# B&R Automation Studio project perfxxl
Automation Studio 4.1.4.402

## Configuration Config1

CPU , AutomationRuntime A3.10, Build 2.95.3, Vc V4.14.1

### Task classes (Cpu.sw)
```
Cyclic#1 (cycle 1000 us, tolerance 40000 us):
  flow <- Processor.flow.prg
Cyclic#2 (cycle 5000 us, tolerance 5000000 us):
  lccount <- Processor.lccount.prg
  seriell <- Exposer.Hardware.seriell.prg
  in_out <- Exposer.Hardware.in_out.prg
  papentf <- Exposer.Ablauf.papentf.prg
  aufnahme <- Exposer.Ablauf.aufnahme.prg
  adjust <- Exposer.Ablauf.adjust.prg
  entladen <- Exposer.Ablauf.entladen.prg
  can_comm <- Exposer.Hardware.can_comm.prg
  expose <- Exposer.Ablauf.expose.prg
  egmio <- Processor.egmio.prg
Cyclic#3 (cycle 10000 us, tolerance 5000000 us):
  lust_cdd <- Exposer.Hardware.lust_cdd.prg
  ip_srv_c <- ip_srv_c.prg
  motors <- Processor.motors.prg
  preheat <- Processor.preheat.prg
Cyclic#4 (cycle 40000 us, tolerance 4000000 us):
  pics <- Visualisierung.pics.prg
  sram <- sram.prg
  p_achse <- Visualisierung.p_achse.prg
  motoren <- Exposer.Hardware.motoren.prg
  trolley <- Exposer.Ablauf.trolley.prg
  ip_clt_c <- ip_clt_c.prg
  referenz <- Exposer.Ablauf.referenz.prg
  system <- system.prg
  devtank <- Processor.devtank.prg
  egmauto <- Processor.egmauto.prg
Cyclic#5 (cycle 100000 us, tolerance 10000000 us):
  file <- file.prg
  xml <- xml.prg
  bluefin <- bluefin.prg
  egmser <- Processor.egmser.prg [disabled]
  tanks <- Processor.tanks.prg
  hwconfig <- hwconfig.prg
  udp_nl <- udp_nl.prg
DataObjects: ioimgcfg <- Datenobj.ioimgcfg.dob, can_tab <- Datenobj.can_tab.dob, do_ima <- Datenobj.do_ima.dob, do_vcp <- Datenobj.do_vcp.dob, do_xsold <- Datenobj.do_xsold.dob
VcDataObjects: visual <- Visualisierung.visual.dob
Binaries: iomap2, iomap1, arcfg2, arcfg1, AsHW, sysconf, vcbmpng
Libraries: visapi, sys_lib, standard, runtime, OPERATOR, LoopCont, INACLNT, FileIO, EthSock, Ethernet, dvframe, DataObj, CONVERT, CAN_Lib, brsystem, AsUDP, AsTime, AsString, AsIOMMan, AsIMA, AsARCfg
```

### Hardware
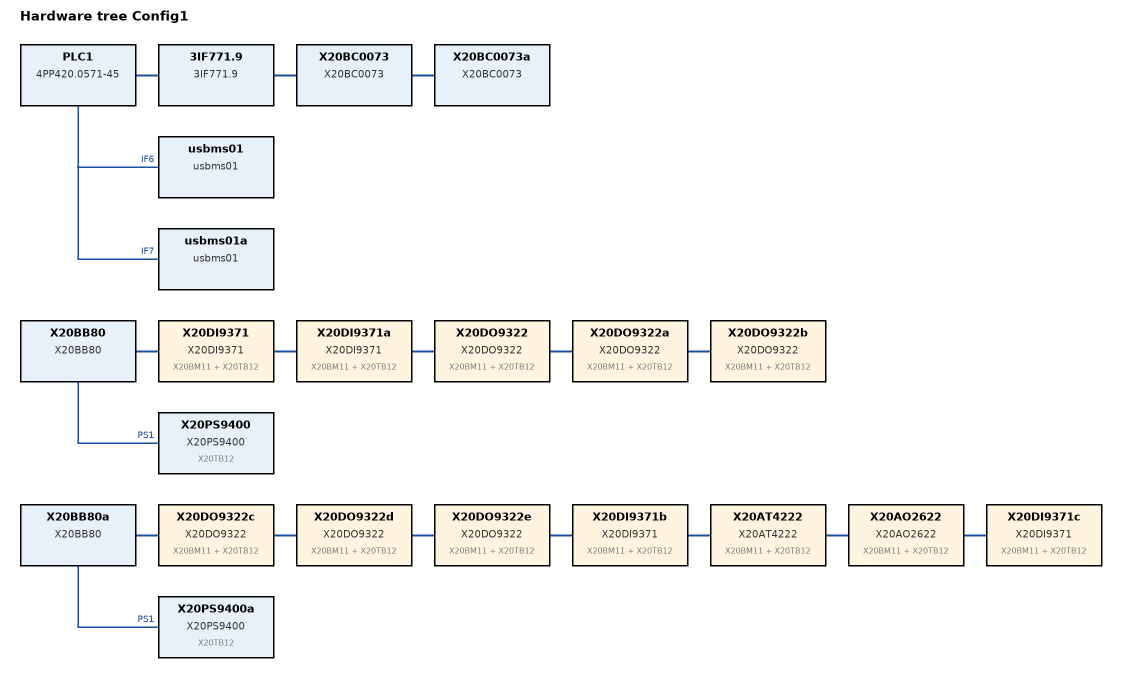
```
3IF771.9 : 3IF771.9 v1.0.2.1  [SS -> PLC1.SS1]
  Connector IF1:
    Baudrate = 250000
    ActivateIna = 1
PLC1 : 4PP420.0571-45 v1.0.0.0
  Connector IF5:
    ActivateDevice = 1
    Mode = Manual
    InternetAddress = 192.168.77.100
    SubnetMask = 255.255.255.0
    Vnc1
    VncVcObjectName1 = visual
    VncKeyMappingFile1 = VCPS2_Keyboard.dis
    VncAuthentication1 = 1
    VncPasswordViewControl1 = laser
    VncMaxConnections1 = 4
  PermanentPvSize = 30000
  RemanentGlobalPvSize = 30000
  VolatileGlobalPvSize = 20000
  PreservePermanentPvMemory = 1
  BRObjects = 400
  Connections = 8
  XLinkUseDefault = 0
  Cyclic1Duration = 1000
  Cyclic1Tolerance = 40000
  Cyclic2Duration = 5000
  Cyclic2Tolerance = 5000000
  Cyclic3Duration = 10000
  Cyclic3Tolerance = 5000000
  Cyclic4Duration = 40000
  Cyclic4Tolerance = 4000000
  Cyclic5Duration = 100000
  Cyclic5Tolerance = 10000000
  Cyclic6Duration = 500000
  Cyclic6Tolerance = 500000
  Cyclic7Duration = 1000000
  Cyclic7Tolerance = 1000000
  Cyclic8Duration = 10000
  Cyclic8Tolerance = 30000000
  FileDevice1
  FileDeviceName1 = DATA
  FileDevicePath1 = C:\USER\
  FileDevice2
  FileDeviceName2 = ROOT
  FileDevicePath2 = C:\
  FileDevice3
  FileDeviceName3 = USBStick
  FileDevicePath3 = IF6.ST1
  FileDevice4
  FileDeviceName4 = USBStick2
  FileDevicePath4 = IF7.ST1
  EthernetHostName = BR_HOST
  EthernetDefaultGateway = 255.255.255.255
  ActivateWebServer = 0
  ActivateSdm = 0
  VcObjectName = visual
usbms01 : usbms01 v1.0.0.0  [USB1 -> PLC1.IF6]
usbms01a : usbms01 v1.0.0.0  [USB1 -> PLC1.IF7]
X20AO2622 : X20AO2622 v1.0.3.0  [SS1 -> X20TB12k.SS; SL -> X20BM11j.SL1]
  FunctionModel = CANIOBusController
  Supervision = off
X20AT4222 : X20AT4222 v1.0.5.0  [SS1 -> X20TB12j.SS; SL -> X20BM11i.SL1]
  FunctionModel = CANIOBusController
  Supervision = off
X20BB80 : X20BB80 v1.0.0.2
X20BB80a : X20BB80 v1.0.0.2
X20BC0073 : X20BC0073 v1.0.3.1  [CAN1 -> 3IF771.9.IF1 (NodeNumber=1); SL -> X20BB80.SL1]
X20BC0073a : X20BC0073 v1.0.3.1  [CAN1 -> X20BC0073.CAN2 (NodeNumber=2); SL -> X20BB80a.SL1]
  InhibitTimeDI = 1
X20BM11 : X20BM11 v1.0.0.0  [X2X1 -> X20BB80.IF1]
X20BM11a : X20BM11 v1.0.0.0  [X2X1 -> X20BM11.X2X2]
X20BM11b : X20BM11 v1.0.0.0  [X2X1 -> X20BM11a.X2X2]
X20BM11c : X20BM11 v1.0.0.0  [X2X1 -> X20BM11b.X2X2]
X20BM11d : X20BM11 v1.0.0.0  [X2X1 -> X20BM11c.X2X2]
X20BM11e : X20BM11 v1.0.0.0  [X2X1 -> X20BB80a.IF1]
X20BM11f : X20BM11 v1.0.0.0  [X2X1 -> X20BM11e.X2X2]
X20BM11g : X20BM11 v1.0.0.0  [X2X1 -> X20BM11f.X2X2]
X20BM11h : X20BM11 v1.0.0.0  [X2X1 -> X20BM11g.X2X2]
X20BM11i : X20BM11 v1.0.0.0  [X2X1 -> X20BM11h.X2X2]
X20BM11j : X20BM11 v1.0.0.0  [X2X1 -> X20BM11i.X2X2]
X20BM11k : X20BM11 v1.0.0.0  [X2X1 -> X20BM11j.X2X2]
X20DI9371 : X20DI9371 v1.0.1.1  [SS1 -> X20TB12.SS; SL -> X20BM11.SL1]
  FunctionModel = CANIOBusController
  Supervision = off
X20DI9371a : X20DI9371 v1.0.1.1  [SS1 -> X20TB12a.SS; SL -> X20BM11a.SL1]
  FunctionModel = CANIOBusController
  Supervision = off
X20DI9371b : X20DI9371 v1.0.1.1  [SS1 -> X20TB12i.SS; SL -> X20BM11h.SL1]
  FunctionModel = CANIOBusController
  Supervision = off
X20DI9371c : X20DI9371 v1.0.1.1  [SS1 -> X20TB12l.SS; SL -> X20BM11k.SL1]
  FunctionModel = CANIOBusController
  Supervision = off
  InputFilter = 2
X20DO9322 : X20DO9322 v1.0.2.2  [SS1 -> X20TB12b.SS; SL -> X20BM11b.SL1]
  FunctionModel = CANIOBusController
  Supervision = off
X20DO9322a : X20DO9322 v1.0.2.2  [SS1 -> X20TB12c.SS; SL -> X20BM11c.SL1]
  FunctionModel = CANIOBusController
  Supervision = off
X20DO9322b : X20DO9322 v1.0.2.2  [SS1 -> X20TB12d.SS; SL -> X20BM11d.SL1]
  FunctionModel = CANIOBusController
  Supervision = off
X20DO9322c : X20DO9322 v1.0.2.2  [SS1 -> X20TB12f.SS; SL -> X20BM11e.SL1]
  FunctionModel = CANIOBusController
  Supervision = off
X20DO9322d : X20DO9322 v1.0.2.2  [SS1 -> X20TB12g.SS; SL -> X20BM11f.SL1]
  FunctionModel = CANIOBusController
  Supervision = off
X20DO9322e : X20DO9322 v1.0.2.2  [SS1 -> X20TB12h.SS; SL -> X20BM11g.SL1]
  FunctionModel = CANIOBusController
  Supervision = off
X20PS9400 : X20PS9400 v1.0.2.0  [SS1 -> X20TB12e.SS; PS -> X20BB80.PS1]
  FunctionModel = CANIOBusController
  Supervision = off
X20PS9400a : X20PS9400 v1.0.2.0  [SS1 -> X20TB12m.SS; PS -> X20BB80a.PS1]
  FunctionModel = CANIOBusController
  Supervision = off
X20TB12 : X20TB12 v1.0.0.0
X20TB12a : X20TB12 v1.0.0.0
X20TB12b : X20TB12 v1.0.0.0
X20TB12c : X20TB12 v1.0.0.0
X20TB12d : X20TB12 v1.0.0.0
X20TB12e : X20TB12 v1.0.0.0
X20TB12f : X20TB12 v1.0.0.0
X20TB12g : X20TB12 v1.0.0.0
X20TB12h : X20TB12 v1.0.0.0
X20TB12i : X20TB12 v1.0.0.0
X20TB12j : X20TB12 v1.0.0.0
X20TB12k : X20TB12 v1.0.0.0
X20TB12l : X20TB12 v1.0.0.0
X20TB12m : X20TB12 v1.0.0.0
```

### Cpu.per - PLC1/Cpu.per
```iecst
(********************************************************************
 * COPYRIGHT --
 ********************************************************************
 * Datei: Cpu.per
 * Autor: Aden
 * Erstellt: 22. Januar 2016
 ********************************************************************
 * Deklaration der permanenten Variablen
 ********************************************************************)
VAR_CONFIG
	DeveloperChangeDate AT %MD25000; (* *)
	IOChangeStep AT %MB25077; (* *)
	IOConfiguration AT %MB25076; (* 1=standard, 2=1250 zus. Temp.Modul *)
	OverallPlateCounter AT %MD25004; (* *)
	OverallReplenisherCounter AT %MD25008; (* *)
	OverallReplenisherPumpTime AT %MD25012; (* *)
	OverallSqmCounter AT %MD25016; (* *)
	ReplenisherCounter AT %MD25060; (* *)
	ReplenisherUsedSinceDevChg AT %MD25064; (* *)
	SRAM AT %MB0; (* *)
	ShutDownTime AT %MD25072; (* *)
	SqmSinceDevChg AT %MD25068; (* *)
	dummy AT %MB25020; (* *)
END_VAR
```

### IoMap.iom - PLC1/IoMap.iom
```iecst
(********************************************************************

	 * COPYRIGHT -- Bernecker & Rainer

	 ********************************************************************

	 * File: IOMap.iom

	 * Author: Aden

	 * Created: 12.09.2005

	 ********************************************************************

	 * IO mapping file

	 ********************************************************************)
VAR_CONFIG
	Cyclic#1.CPUTemp AT %IW."PLC1".TemperatureCPU;
	Cyclic#1.AmbientTemp AT %IW."PLC1".TemperatureENV;
	Cyclic#1.BatteryStatus AT %IB."PLC1".BatteryStatusCPU;
	Cyclic#1.egmio:EGMModule1Out[0] AT %QX."X20DO9322c".DigitalOutput01;
	Cyclic#1.egmio:EGMModule1Out[1] AT %QX."X20DO9322c".DigitalOutput02;
	Cyclic#1.egmio:EGMModule1Out[2] AT %QX."X20DO9322c".DigitalOutput03;
	Cyclic#1.egmio:EGMModule1Out[3] AT %QX."X20DO9322c".DigitalOutput04;
	Cyclic#1.egmio:EGMModule1Out[4] AT %QX."X20DO9322c".DigitalOutput05;
	Cyclic#1.egmio:EGMModule1Out[5] AT %QX."X20DO9322c".DigitalOutput06;
	Cyclic#1.egmio:EGMModule1Out[6] AT %QX."X20DO9322c".DigitalOutput07;
	Cyclic#1.egmio:EGMModule1Out[7] AT %QX."X20DO9322c".DigitalOutput08;
	Cyclic#1.egmio:EGMModule1Out[8] AT %QX."X20DO9322c".DigitalOutput09;
	Cyclic#1.egmio:EGMModule1Out[9] AT %QX."X20DO9322c".DigitalOutput10;
	Cyclic#1.egmio:EGMModule1Out[10] AT %QX."X20DO9322c".DigitalOutput11;
	Cyclic#1.egmio:EGMModule1Out[11] AT %QX."X20DO9322c".DigitalOutput12;
	ModulStatus_DO1 AT %IX."X20DO9322c".ModuleOk;
	ModulStatus_DO2 AT %IX."X20DO9322d".ModuleOk;
	Cyclic#1.egmio:EGMModule2Out[0] AT %QX."X20DO9322d".DigitalOutput01;
	Cyclic#1.egmio:EGMModule2Out[1] AT %QX."X20DO9322d".DigitalOutput02;
	Cyclic#1.egmio:EGMModule2Out[2] AT %QX."X20DO9322d".DigitalOutput03;
	Cyclic#1.egmio:EGMModule2Out[3] AT %QX."X20DO9322d".DigitalOutput04;
	Cyclic#1.egmio:EGMModule2Out[4] AT %QX."X20DO9322d".DigitalOutput05;
	Cyclic#1.egmio:EGMModule2Out[5] AT %QX."X20DO9322d".DigitalOutput06;
	Cyclic#1.egmio:EGMModule2Out[6] AT %QX."X20DO9322d".DigitalOutput07;
	ModulStatus_DO3 AT %IX."X20DO9322e".ModuleOk;
	Cyclic#1.egmio:EGMModule3Out[0] AT %QX."X20DO9322e".DigitalOutput01;
	Cyclic#1.egmio:EGMModule3Out[1] AT %QX."X20DO9322e".DigitalOutput02;
	Cyclic#1.egmio:EGMModule3Out[2] AT %QX."X20DO9322e".DigitalOutput03;
	Cyclic#1.egmio:EGMModule3Out[3] AT %QX."X20DO9322e".DigitalOutput04;
	Cyclic#1.egmio:EGMModule3Out[4] AT %QX."X20DO9322e".DigitalOutput05;
	Cyclic#1.egmio:EGMModule3Out[5] AT %QX."X20DO9322e".DigitalOutput06;
	Cyclic#1.egmio:EGMModule3Out[6] AT %QX."X20DO9322e".DigitalOutput07;
	Cyclic#1.egmio:EGMModule3Out[7] AT %QX."X20DO9322e".DigitalOutput08;
	Cyclic#1.ModulStatus_DI AT %IX."X20DI9371b".ModuleOk;
	Cyclic#1.egmio:EGMModule1In[0] AT %IX."X20DI9371b".DigitalInput01;
	Cyclic#1.egmio:EGMModule1In[1] AT %IX."X20DI9371b".DigitalInput02;
	Cyclic#1.egmio:EGMModule1In[2] AT %IX."X20DI9371b".DigitalInput03;
	Cyclic#1.egmio:EGMModule1In[3] AT %IX."X20DI9371b".DigitalInput04;
	Cyclic#1.egmio:EGMModule1In[4] AT %IX."X20DI9371b".DigitalInput05;
	Cyclic#1.egmio:EGMModule1In[5] AT %IX."X20DI9371b".DigitalInput06;
	Cyclic#1.egmio:EGMModule1In[6] AT %IX."X20DI9371b".DigitalInput07;
	Cyclic#1.egmio:EGMModule1In[7] AT %IX."X20DI9371b".DigitalInput08;
	Cyclic#1.egmio:EGMModule1In[8] AT %IX."X20DI9371b".DigitalInput09;
	Cyclic#1.egmio:EGMModule1In[9] AT %IX."X20DI9371b".DigitalInput10;
	Cyclic#1.ModulStatus_AT AT %IX."X20AT4222".ModuleOk;
	Cyclic#1.EGMPreheat.AmbientTemp[0] AT %IW."X20AT4222".Temperature01;
	Cyclic#1.devtank:TempSensorValue AT %IW."X20AT4222".Temperature02;
	Cyclic#1.ModulStatus_AT1 AT %IB."X20AT4222".StatusInput01;
	ModulStatus_AO AT %IX."X20AO2622".ModuleOk;
	Cyclic#1.EGMMainMotor.RatedRpm AT %QW."X20AO2622".AnalogOutput01;
	Cyclic#1.EGMBrushMotor.RatedRpm AT %QW."X20AO2622".AnalogOutput02;
	Cyclic#1.ModulStatus_PS AT %IX."X20PS9400a".ModuleOk;
	Cyclic#1.ModulStatus_PS1 AT %IX."X20PS9400a".StatusInput01;
	Cyclic#1.ModulStatus_PS2 AT %IX."X20PS9400a".StatusInput02;
	Cyclic#1.ModulStatus_DI2 AT %IX."X20DI9371c".ModuleOk;
	Cyclic#1.egmio:EGMModule2In[0] AT %IX."X20DI9371c".DigitalInput01;
	Cyclic#1.egmio:EGMModule2In[1] AT %IX."X20DI9371c".DigitalInput02;
	Cyclic#1.egmio:EGMModule2In[2] AT %IX."X20DI9371c".DigitalInput03;
	Cyclic#1.egmio:EGMModule2In[3] AT %IX."X20DI9371c".DigitalInput04;
	Cyclic#1.egmio:EGMModule2In[4] AT %IX."X20DI9371c".DigitalInput05;
	Cyclic#1.egmio:EGMModule2In[5] AT %IX."X20DI9371c".DigitalInput06;
	Cyclic#1.EGMPreheat.RealTemp[0] AT %IW."X20AT4222".Temperature03;
	Cyclic#1.EGMPreheat.RealTemp[1] AT %IW."X20AT4222".Temperature04;
	Cyclic#1.egmio:EGMModule1In[10] AT %IX."X20DI9371b".DigitalInput11;
	Cyclic#1.egmio:EGMModule2Out[7] AT %QX."X20DO9322d".DigitalOutput08;
	Cyclic#1.egmio:EGMModule2Out[8] AT %QX."X20DO9322d".DigitalOutput09;
	Cyclic#1.egmio:EGMModule2Out[9] AT %QX."X20DO9322d".DigitalOutput10;
	Cyclic#1.egmio:EGMModule2Out[10] AT %QX."X20DO9322d".DigitalOutput11;
	Cyclic#1.egmio:EGMModule2Out[11] AT %QX."X20DO9322d".DigitalOutput12;
	Cyclic#1.egmio:EGMModule3Out[8] AT %QX."X20DO9322e".DigitalOutput09;
	Cyclic#1.egmio:EGMModule3Out[9] AT %QX."X20DO9322e".DigitalOutput10;
	Cyclic#1.egmio:EGMModule3Out[10] AT %QX."X20DO9322e".DigitalOutput11;
	Cyclic#1.egmio:EGMModule3Out[11] AT %QX."X20DO9322e".DigitalOutput12;
	Cyclic#1.egmio:EGMModule1In[11] AT %IX."X20DI9371b".DigitalInput12;
	Cyclic#1.egmio:EGMModule2In[6] AT %IX."X20DI9371c".DigitalInput07;
	Cyclic#1.egmio:EGMModule2In[7] AT %IX."X20DI9371c".DigitalInput08;
	Cyclic#1.egmio:EGMModule2In[8] AT %IX."X20DI9371c".DigitalInput09;
	Cyclic#1.egmio:EGMModule2In[9] AT %IX."X20DI9371c".DigitalInput10;
	Cyclic#1.egmio:EGMModule2In[10] AT %IX."X20DI9371c".DigitalInput11;
	Cyclic#1.egmio:EGMModule2In[11] AT %IX."X20DI9371c".DigitalInput12;
	Cyclic#1.CANNodeNumber AT %IB."3IF771.9".IF1.NodeSwitch;
	Cyclic#1.In_ServiceMode AT %IX."X20DI9371".DigitalInput01;
	Cyclic#1.In_PaperSensor[0] AT %IX."X20DI9371".DigitalInput03;
	Cyclic#1.In_PaperSensor[1] AT %IX."X20DI9371".DigitalInput04;
	Cyclic#1.In_FeederHorActive AT %IX."X20DI9371".DigitalInput05;
	Cyclic#1.In_FeederHorInactive AT %IX."X20DI9371".DigitalInput06;
	Cyclic#1.In_FeederVacuumOK[0] AT %IX."X20DI9371".DigitalInput07;
	Cyclic#1.In_FeederVacuumOK[1] AT %IX."X20DI9371".DigitalInput08;
	Cyclic#1.In_FeederVacuumOK[2] AT %IX."X20DI9371".DigitalInput09;
	Cyclic#1.In_FeederVacuumOK[3] AT %IX."X20DI9371".DigitalInput10;
	Cyclic#1.In_FeederVacuumOK[4] AT %IX."X20DI9371".DigitalInput11;
	Cyclic#1.In_FeederVacuumOK[5] AT %IX."X20DI9371".DigitalInput12;
	Cyclic#1.In_PlateAdjusted[0] AT %IX."X20DI9371a".DigitalInput01;
	Cyclic#1.In_PlateAdjusted[1] AT %IX."X20DI9371a".DigitalInput02;
	Cyclic#1.In_LiftingPinsDown AT %IX."X20DI9371a".DigitalInput03;
	Cyclic#1.In_ConveyorBeltSensor[0] AT %IX."X20DI9371a".DigitalInput04 INVERSE;
	Cyclic#1.In_ConveyorBeltSensor[1] AT %IX."X20DI9371a".DigitalInput05 INVERSE;
	Cyclic#1.TrolleyCodeSensor AT %IX."X20DI9371a".DigitalInput07;
	Cyclic#1.BeltLoose AT %IX."X20DI9371a".DigitalInput08;
	Cyclic#1.in_out:Module4[0] AT %QX."X20DO9322".DigitalOutput01;
	Cyclic#1.in_out:Module4[1] AT %QX."X20DO9322".DigitalOutput02;
	Cyclic#1.in_out:Module4[2] AT %QX."X20DO9322".DigitalOutput03;
	Cyclic#1.in_out:Module4[3] AT %QX."X20DO9322".DigitalOutput04;
	Cyclic#1.in_out:Module4[4] AT %QX."X20DO9322".DigitalOutput05;
	Cyclic#1.in_out:Module4[5] AT %QX."X20DO9322".DigitalOutput06;
	Cyclic#1.in_out:Module4[6] AT %QX."X20DO9322".DigitalOutput07;
	Cyclic#1.in_out:Module4[7] AT %QX."X20DO9322".DigitalOutput08;
	Cyclic#1.in_out:Module4[8] AT %QX."X20DO9322".DigitalOutput09;
	Cyclic#1.in_out:Module4[9] AT %QX."X20DO9322".DigitalOutput10;
	Cyclic#1.in_out:Module4[10] AT %QX."X20DO9322".DigitalOutput11;
	Cyclic#1.in_out:Module4[11] AT %QX."X20DO9322".DigitalOutput12;
	Cyclic#1.in_out:Module5[0] AT %QX."X20DO9322a".DigitalOutput01;
	Cyclic#1.in_out:Module5[1] AT %QX."X20DO9322a".DigitalOutput02;
	Cyclic#1.in_out:Module5[2] AT %QX."X20DO9322a".DigitalOutput03;
	Cyclic#1.in_out:Module5[3] AT %QX."X20DO9322a".DigitalOutput04;
	Cyclic#1.in_out:Module5[4] AT %QX."X20DO9322a".DigitalOutput05;
	Cyclic#1.in_out:Module5[5] AT %QX."X20DO9322a".DigitalOutput06;
	Cyclic#1.in_out:Module5[6] AT %QX."X20DO9322a".DigitalOutput07;
	Cyclic#1.in_out:Module5[7] AT %QX."X20DO9322a".DigitalOutput08;
	Cyclic#1.in_out:Module5[8] AT %QX."X20DO9322a".DigitalOutput09;
	Cyclic#1.in_out:Module5[9] AT %QX."X20DO9322a".DigitalOutput10;
	Cyclic#1.in_out:Module5[10] AT %QX."X20DO9322a".DigitalOutput11;
	Cyclic#1.in_out:Module5[11] AT %QX."X20DO9322a".DigitalOutput12;
	Cyclic#1.in_out:Module6[0] AT %QX."X20DO9322b".DigitalOutput01;
	Cyclic#1.in_out:Module6[1] AT %QX."X20DO9322b".DigitalOutput02;
	Cyclic#1.in_out:Module6[2] AT %QX."X20DO9322b".DigitalOutput03;
	Cyclic#1.in_out:Module6[3] AT %QX."X20DO9322b".DigitalOutput04;
	Cyclic#1.in_out:Module6[4] AT %QX."X20DO9322b".DigitalOutput05;
	Cyclic#1.in_out:Module6[5] AT %QX."X20DO9322b".DigitalOutput06;
	Cyclic#1.in_out:Module6[6] AT %QX."X20DO9322b".DigitalOutput07;
	Cyclic#1.in_out:Module6[7] AT %QX."X20DO9322b".DigitalOutput08;
	Cyclic#1.in_out:Module6[8] AT %QX."X20DO9322b".DigitalOutput09;
	Cyclic#1.in_out:Module6[9] AT %QX."X20DO9322b".DigitalOutput10;
	Cyclic#1.in_out:Module6[10] AT %QX."X20DO9322b".DigitalOutput11;
	Cyclic#1.in_out:Module6[11] AT %QX."X20DO9322b".DigitalOutput12;
	Cyclic#1.CoverLockOK AT %IX."X20DI9371a".DigitalInput09;
	Cyclic#1.DoorsOK AT %IX."X20DI9371a".DigitalInput10;
END_VAR
```

### Beide.osl - PLC1/States/Beide.osl
```
ObjectStates:
  Object flow (Memory=UserROM, Enable=true)
  Object lccount (Memory=UserROM, Enable=true)
  Object seriell (Memory=UserROM, Enable=true)
  Object in_out (Memory=UserROM, Enable=true)
  Object papentf (Memory=UserROM, Enable=true)
  Object aufnahme (Memory=UserROM, Enable=true)
  Object adjust (Memory=UserROM, Enable=true)
  Object entladen (Memory=UserROM, Enable=true)
  Object can_comm (Memory=UserROM, Enable=true)
  Object expose (Memory=UserROM, Enable=true)
  Object egmio (Memory=UserROM, Enable=true)
  Object lust_cdd (Memory=UserROM, Enable=true)
  Object ip_srv_c (Memory=UserROM, Enable=true)
  Object motors (Memory=UserROM, Enable=true)
  Object preheat (Memory=UserROM, Enable=true)
  Object pics (Memory=UserROM, Enable=true)
  Object sram (Memory=UserROM, Enable=true)
  Object p_achse (Memory=UserROM, Enable=true)
  Object motoren (Memory=UserROM, Enable=true)
  Object trolley (Memory=UserROM, Enable=true)
  Object ip_clt_c (Memory=UserROM, Enable=true)
  Object referenz (Memory=UserROM, Enable=true)
  Object system (Memory=UserROM, Enable=true)
  Object devtank (Memory=UserROM, Enable=true)
  Object egmauto (Memory=UserROM, Enable=true)
  Object file (Memory=UserROM, Enable=true)
  Object xml (Memory=UserROM, Enable=true)
  Object bluefin (Memory=UserROM, Enable=true)
  Object egmser (Memory=UserROM, Enable=false)
  Object tanks (Memory=UserROM, Enable=true)
  Object hwconfig (Memory=UserROM, Enable=true)
  Object udp_nl (Memory=UserROM, Enable=true)
  Object ioimgcfg (Memory=UserROM, Enable=true)
  Object can_tab (Memory=UserROM, Enable=true)
  Object do_ima (Memory=UserROM, Enable=true)
  Object do_vcp (Memory=UserROM, Enable=true)
  Object do_xsold (Memory=UserROM, Enable=true)
  Object visual (Memory=UserROM, Enable=true)
  Object iomap2 (Memory=UserROM, Enable=true)
  Object iomap1 (Memory=UserROM, Enable=true)
  Object arcfg2 (Memory=UserROM, Enable=true)
  Object arcfg1 (Memory=UserROM, Enable=true)
  Object AsHW (Memory=UserROM, Enable=true)
  Object sysconf (Memory=SystemROM, Enable=true)
  Object vcbmpng (Memory=UserROM, Enable=true)
```

### Bluefin.osl - PLC1/States/Bluefin.osl
```
ObjectStates:
  Object flow (Memory=UserROM, Enable=true)
  Object lccount (Memory=UserROM, Enable=true)
  Object seriell (Memory=UserROM, Enable=false)
  Object in_out (Memory=UserROM, Enable=false)
  Object papentf (Memory=UserROM, Enable=false)
  Object aufnahme (Memory=UserROM, Enable=false)
  Object adjust (Memory=UserROM, Enable=false)
  Object entladen (Memory=UserROM, Enable=false)
  Object can_comm (Memory=UserROM, Enable=false)
  Object expose (Memory=UserROM, Enable=false)
  Object egmio (Memory=UserROM, Enable=true)
  Object lust_cdd (Memory=UserROM, Enable=false)
  Object ip_srv_c (Memory=UserROM, Enable=false)
  Object motors (Memory=UserROM, Enable=true)
  Object preheat (Memory=UserROM, Enable=true)
  Object pics (Memory=UserROM, Enable=true)
  Object sram (Memory=UserROM, Enable=true)
  Object p_achse (Memory=UserROM, Enable=false)
  Object motoren (Memory=UserROM, Enable=false)
  Object trolley (Memory=UserROM, Enable=false)
  Object ip_clt_c (Memory=UserROM, Enable=false)
  Object referenz (Memory=UserROM, Enable=false)
  Object system (Memory=UserROM, Enable=true)
  Object devtank (Memory=UserROM, Enable=true)
  Object egmauto (Memory=UserROM, Enable=true)
  Object file (Memory=UserROM, Enable=true)
  Object xml (Memory=UserROM, Enable=true)
  Object bluefin (Memory=UserROM, Enable=false)
  Object egmser (Memory=UserROM, Enable=true)
  Object tanks (Memory=UserROM, Enable=true)
  Object hwconfig (Memory=UserROM, Enable=true)
  Object udp_nl (Memory=UserROM, Enable=true)
  Object ioimgcfg (Memory=UserROM, Enable=true)
  Object can_tab (Memory=UserROM, Enable=true)
  Object do_ima (Memory=UserROM, Enable=true)
  Object do_vcp (Memory=UserROM, Enable=true)
  Object do_xsold (Memory=UserROM, Enable=true)
  Object visual (Memory=UserROM, Enable=true)
  Object iomap2 (Memory=UserROM, Enable=true)
  Object iomap1 (Memory=UserROM, Enable=true)
  Object arcfg2 (Memory=UserROM, Enable=true)
  Object arcfg1 (Memory=UserROM, Enable=true)
  Object AsHW (Memory=UserROM, Enable=true)
  Object sysconf (Memory=SystemROM, Enable=true)
  Object vcbmpng (Memory=UserROM, Enable=true)
```

### Performance.osl - PLC1/States/Performance.osl
```
ObjectStates:
  Object flow (Memory=UserROM, Enable=false)
  Object lccount (Memory=UserROM, Enable=false)
  Object seriell (Memory=UserROM, Enable=true)
  Object in_out (Memory=UserROM, Enable=true)
  Object papentf (Memory=UserROM, Enable=true)
  Object aufnahme (Memory=UserROM, Enable=true)
  Object adjust (Memory=UserROM, Enable=true)
  Object entladen (Memory=UserROM, Enable=true)
  Object can_comm (Memory=UserROM, Enable=true)
  Object expose (Memory=UserROM, Enable=true)
  Object egmio (Memory=UserROM, Enable=false)
  Object lust_cdd (Memory=UserROM, Enable=true)
  Object ip_srv_c (Memory=UserROM, Enable=true)
  Object motors (Memory=UserROM, Enable=false)
  Object preheat (Memory=UserROM, Enable=false)
  Object pics (Memory=UserROM, Enable=true)
  Object sram (Memory=UserROM, Enable=true)
  Object p_achse (Memory=UserROM, Enable=true)
  Object motoren (Memory=UserROM, Enable=true)
  Object trolley (Memory=UserROM, Enable=true)
  Object ip_clt_c (Memory=UserROM, Enable=true)
  Object referenz (Memory=UserROM, Enable=true)
  Object system (Memory=UserROM, Enable=true)
  Object devtank (Memory=UserROM, Enable=false)
  Object egmauto (Memory=UserROM, Enable=false)
  Object file (Memory=UserROM, Enable=true)
  Object xml (Memory=UserROM, Enable=false)
  Object bluefin (Memory=UserROM, Enable=true)
  Object egmser (Memory=UserROM, Enable=false)
  Object tanks (Memory=UserROM, Enable=false)
  Object hwconfig (Memory=UserROM, Enable=true)
  Object udp_nl (Memory=UserROM, Enable=true)
  Object ioimgcfg (Memory=UserROM, Enable=true)
  Object can_tab (Memory=UserROM, Enable=true)
  Object do_ima (Memory=UserROM, Enable=true)
  Object do_vcp (Memory=UserROM, Enable=true)
  Object do_xsold (Memory=UserROM, Enable=true)
  Object visual (Memory=UserROM, Enable=true)
  Object iomap2 (Memory=UserROM, Enable=true)
  Object iomap1 (Memory=UserROM, Enable=true)
  Object arcfg2 (Memory=UserROM, Enable=true)
  Object arcfg1 (Memory=UserROM, Enable=true)
  Object AsHW (Memory=UserROM, Enable=true)
  Object sysconf (Memory=SystemROM, Enable=true)
  Object vcbmpng (Memory=UserROM, Enable=true)
```

## Configuration PPC2100

CPU 5PPC2100.BY01-000, AutomationRuntime S4.10, Build 4.1.2, Vc V4.15.9

### Task classes (Cpu.sw)
```
Cyclic#1 (cycle 1000 us, tolerance 40000 us):
  flow <- Processor.flow.prg
Cyclic#2 (cycle 5000 us, tolerance 5000000 us):
  lccount <- Processor.lccount.prg
  seriell <- Exposer.Hardware.seriell.prg
  in_out <- Exposer.Hardware.in_out.prg
  papentf <- Exposer.Ablauf.papentf.prg
  aufnahme <- Exposer.Ablauf.aufnahme.prg
  adjust <- Exposer.Ablauf.adjust.prg
  entladen <- Exposer.Ablauf.entladen.prg
  can_comm <- Exposer.Hardware.can_comm.prg
  expose <- Exposer.Ablauf.expose.prg
  egmio <- Processor.egmio.prg
Cyclic#3 (cycle 10000 us, tolerance 5000000 us):
  lust_cdd <- Exposer.Hardware.lust_cdd.prg
  ip_srv_c <- ip_srv_c.prg
  motors <- Processor.motors.prg
  preheat <- Processor.preheat.prg
Cyclic#4 (cycle 40000 us, tolerance 4000000 us):
  pics <- Visualisierung.pics.prg
  sram <- sram.prg
  p_achse <- Visualisierung.p_achse.prg
  motoren <- Exposer.Hardware.motoren.prg
  trolley <- Exposer.Ablauf.trolley.prg
  ip_clt_c <- ip_clt_c.prg
  referenz <- Exposer.Ablauf.referenz.prg
  system <- system.prg
  devtank <- Processor.devtank.prg
  egmauto <- Processor.egmauto.prg
Cyclic#5 (cycle 100000 us, tolerance 10000000 us):
  file <- file.prg
  xml <- xml.prg
  bluefin <- bluefin.prg
  egmser <- Processor.egmser.prg [disabled]
  tanks <- Processor.tanks.prg
  hwconfig <- hwconfig.prg
  udp_nl <- udp_nl.prg
VcDataObjects: visuhr <- Visualisierung.visuhr.dob
Binaries: asfw, ashwd, arconfig, pvmap, sysconf
Libraries: ethernet, ethsock, fileio, visapi, asstring, standard, astime, asiomman, dataobj, dvframe, can_lib, asarcfg, brsystem, loopcont, asudp, sys_lib, AsBrStr, AsICMP, runtime, AsUSB
```

### Hardware
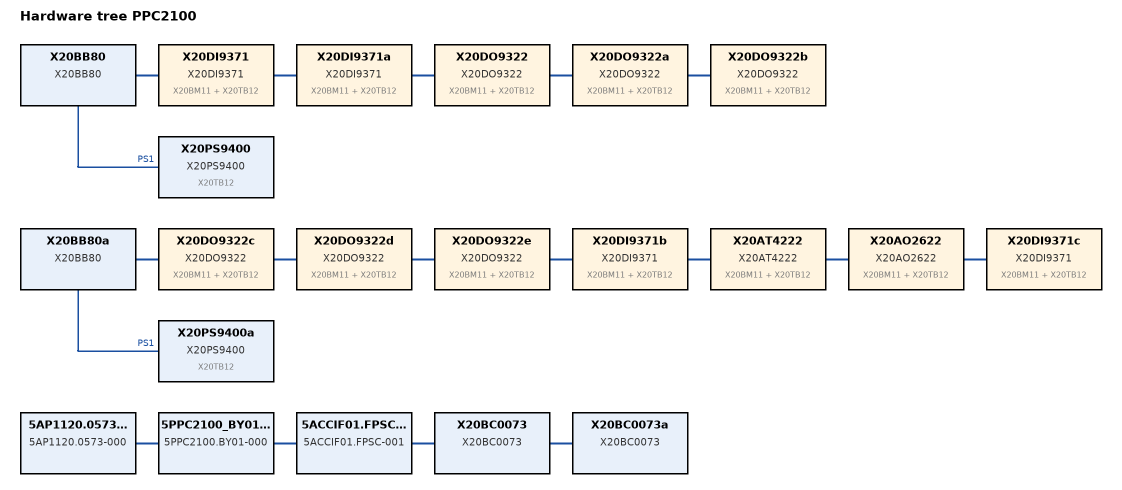
```
5ACCIF01.FPSC-001 : 5ACCIF01.FPSC-001 v1.8.1.0  [SL -> 5PPC2100_BY01_000.SL1]
5AP1120.0573-000 : 5AP1120.0573-000 v2.0.0.0
  VcObjectName = visuhr
5PPC2100_BY01_000 : 5PPC2100.BY01-000 v1.4.0.0  [SY -> 5AP1120.0573-000.SY1]
  Connector IF3:
    ActivateDevice = 1
    Mode = Manual
    Vnc1
    VncVcObjectName1 = visuhr
    VncKeyMappingFile1 = VC\PS2-Keyboard.dis
    VncAuthentication1 = 1
    VncPasswordViewControl1 = laser
    VncMaxConnections1 = 4
    InternetAddress = 192.168.77.100
    SubnetMask = 255.255.255.0
  Connector IF4:
    ActivateDevice = 1
  UserRamDevice = PCI.1.PPC21xx.SRAM
  UserRamSize = 245760
  RemMemDevice = PCI.1.PPC21xx.SRAM
  RemMemSize = 261888
  PermanentPvSize = 30000
  RemanentGlobalPvSize = 30000
  VolatileGlobalPvSize = 20000
  PreservePermanentPvMemory = 1
  BRObjects = 400
  Connections = 8
  Cyclic1Duration = 1000
  Cyclic1Tolerance = 40000
  Cyclic2Duration = 5000
  Cyclic2Tolerance = 5000000
  Cyclic3Duration = 10000
  Cyclic3Tolerance = 5000000
  Cyclic4Duration = 40000
  Cyclic4Tolerance = 4000000
  Cyclic5Duration = 100000
  Cyclic5Tolerance = 10000000
  Cyclic6Duration = 500000
  Cyclic6Tolerance = 500000
  Cyclic7Duration = 1000000
  Cyclic7Tolerance = 1000000
  Cyclic8Duration = 10000
  Cyclic8Tolerance = 30000000
  FileDevice1
  FileDeviceName1 = DATA
  FileDevicePath1 = C:\USER\
  FileDevice2
  FileDeviceName2 = ROOT
  FileDevicePath2 = C:\
  FileDevice3
  EthernetDefaultGateway = 255.255.255.255
  ActivateWebServer = 0
  ActivateSdm = 0
X20AO2622 : X20AO2622 v1.0.3.0  [SS1 -> X20TB12j.SS; SL -> X20BM11h.SL1]
  FunctionModel = CANIOBusController
X20AT4222 : X20AT4222 v1.0.5.0  [SS1 -> X20TB12i.SS; SL -> X20BM11g.SL1]
  FunctionModel = CANIOBusController
X20BB80 : X20BB80 v1.0.0.2
X20BB80a : X20BB80 v1.0.0.2
X20BC0073 : X20BC0073 v1.2.0.0  [CAN1 -> 5ACCIF01.FPSC-001.IF3 (NodeNumber=2); SL -> X20BB80.SL1]
X20BC0073a : X20BC0073 v1.2.0.0  [CAN1 -> X20BC0073.CAN2 (NodeNumber=1); SL -> X20BB80a.SL1]
X20BM11 : X20BM11 v1.0.0.0  [X2X1 -> X20BB80.IF1]
X20BM11a : X20BM11 v1.0.0.0  [X2X1 -> X20BM11b.X2X2]
X20BM11b : X20BM11 v1.0.0.0  [X2X1 -> X20BM11j.X2X2]
X20BM11c : X20BM11 v1.0.0.0  [X2X1 -> X20BM11e.X2X2]
X20BM11d : X20BM11 v1.0.0.0  [X2X1 -> X20BB80a.IF1]
X20BM11e : X20BM11 v1.0.0.0  [X2X1 -> X20BM11d.X2X2]
X20BM11f : X20BM11 v1.0.0.0  [X2X1 -> X20BM11c.X2X2]
X20BM11g : X20BM11 v1.0.0.0  [X2X1 -> X20BM11f.X2X2]
X20BM11h : X20BM11 v1.0.0.0  [X2X1 -> X20BM11g.X2X2]
X20BM11i : X20BM11 v1.0.0.0  [X2X1 -> X20BM11h.X2X2]
X20BM11j : X20BM11 v1.0.0.0  [X2X1 -> X20BM11.X2X2]
X20BM11k : X20BM11 v1.0.0.0  [X2X1 -> X20BM11a.X2X2]
X20DI9371 : X20DI9371 v1.0.1.1  [SS1 -> X20TB12a.SS; SL -> X20BM11.SL1]
  FunctionModel = CANIOBusController
X20DI9371a : X20DI9371 v1.0.1.1  [SS1 -> X20TB12l.SS; SL -> X20BM11j.SL1]
  FunctionModel = CANIOBusController
X20DI9371b : X20DI9371 v1.0.1.1  [SS1 -> X20TB12h.SS; SL -> X20BM11f.SL1]
  FunctionModel = CANIOBusController
X20DI9371c : X20DI9371 v1.0.1.1  [SS1 -> X20TB12k.SS; SL -> X20BM11i.SL1]
  FunctionModel = CANIOBusController
X20DO9322 : X20DO9322 v1.0.2.2  [SS1 -> X20TB12c.SS; SL -> X20BM11b.SL1]
  FunctionModel = CANIOBusController
X20DO9322a : X20DO9322 v1.0.2.2  [SS1 -> X20TB12b.SS; SL -> X20BM11a.SL1]
  FunctionModel = CANIOBusController
X20DO9322b : X20DO9322 v1.0.2.2  [SS1 -> X20TB12m.SS; SL -> X20BM11k.SL1]
  FunctionModel = CANIOBusController
X20DO9322c : X20DO9322 v1.0.2.2  [SS1 -> X20TB12f.SS; SL -> X20BM11d.SL1]
  FunctionModel = CANIOBusController
X20DO9322d : X20DO9322 v1.0.2.2  [SS1 -> X20TB12g.SS; SL -> X20BM11e.SL1]
  FunctionModel = CANIOBusController
X20DO9322e : X20DO9322 v1.0.2.2  [SS1 -> X20TB12e.SS; SL -> X20BM11c.SL1]
  FunctionModel = CANIOBusController
X20PS9400 : X20PS9400 v1.0.2.0  [SS1 -> X20TB12d.SS; PS -> X20BB80.PS1]
X20PS9400a : X20PS9400 v1.0.2.0  [SS1 -> X20TB12.SS; PS -> X20BB80a.PS1]
X20TB12 : X20TB12 v1.0.0.0
X20TB12a : X20TB12 v1.0.0.0
X20TB12b : X20TB12 v1.0.0.0
X20TB12c : X20TB12 v1.0.0.0
X20TB12d : X20TB12 v1.0.0.0
X20TB12e : X20TB12 v1.0.0.0
X20TB12f : X20TB12 v1.0.0.0
X20TB12g : X20TB12 v1.0.0.0
X20TB12h : X20TB12 v1.0.0.0
X20TB12i : X20TB12 v1.0.0.0
X20TB12j : X20TB12 v1.0.0.0
X20TB12k : X20TB12 v1.0.0.0
X20TB12l : X20TB12 v1.0.0.0
X20TB12m : X20TB12 v1.0.0.0
```

### IoMap.iom - 5PPC2100_BY01_000/IoMap.iom
```iecst
(********************************************************************

	 * COPYRIGHT -- Bernecker & Rainer

	 ********************************************************************

	 * File: IOMap.iom

	 * Author: Aden

	 * Created: 12.09.2005

	 ********************************************************************

	 * IO mapping file

	 ********************************************************************)
VAR_CONFIG
	Cyclic#1.egmio:EGMModule1Out[0] AT %QX."X20DO9322c".DigitalOutput01;
	Cyclic#1.egmio:EGMModule1Out[1] AT %QX."X20DO9322c".DigitalOutput02;
	Cyclic#1.egmio:EGMModule1Out[2] AT %QX."X20DO9322c".DigitalOutput03;
	Cyclic#1.egmio:EGMModule1Out[3] AT %QX."X20DO9322c".DigitalOutput04;
	Cyclic#1.egmio:EGMModule1Out[4] AT %QX."X20DO9322c".DigitalOutput05;
	Cyclic#1.egmio:EGMModule1Out[5] AT %QX."X20DO9322c".DigitalOutput06;
	Cyclic#1.egmio:EGMModule1Out[6] AT %QX."X20DO9322c".DigitalOutput07;
	Cyclic#1.egmio:EGMModule1Out[7] AT %QX."X20DO9322c".DigitalOutput08;
	Cyclic#1.egmio:EGMModule1Out[8] AT %QX."X20DO9322c".DigitalOutput09;
	Cyclic#1.egmio:EGMModule1Out[9] AT %QX."X20DO9322c".DigitalOutput10;
	Cyclic#1.egmio:EGMModule1Out[10] AT %QX."X20DO9322c".DigitalOutput11;
	Cyclic#1.egmio:EGMModule1Out[11] AT %QX."X20DO9322c".DigitalOutput12;
	ModulStatus_DO1 AT %IX."X20DO9322c".ModuleOk;
	ModulStatus_DO2 AT %IX."X20DO9322d".ModuleOk;
	Cyclic#1.egmio:EGMModule2Out[0] AT %QX."X20DO9322d".DigitalOutput01;
	Cyclic#1.egmio:EGMModule2Out[1] AT %QX."X20DO9322d".DigitalOutput02;
	Cyclic#1.egmio:EGMModule2Out[2] AT %QX."X20DO9322d".DigitalOutput03;
	Cyclic#1.egmio:EGMModule2Out[3] AT %QX."X20DO9322d".DigitalOutput04;
	Cyclic#1.egmio:EGMModule2Out[4] AT %QX."X20DO9322d".DigitalOutput05;
	Cyclic#1.egmio:EGMModule2Out[5] AT %QX."X20DO9322d".DigitalOutput06;
	Cyclic#1.egmio:EGMModule2Out[6] AT %QX."X20DO9322d".DigitalOutput07;
	ModulStatus_DO3 AT %IX."X20DO9322e".ModuleOk;
	Cyclic#1.egmio:EGMModule3Out[0] AT %QX."X20DO9322e".DigitalOutput01;
	Cyclic#1.egmio:EGMModule3Out[1] AT %QX."X20DO9322e".DigitalOutput02;
	Cyclic#1.egmio:EGMModule3Out[2] AT %QX."X20DO9322e".DigitalOutput03;
	Cyclic#1.egmio:EGMModule3Out[3] AT %QX."X20DO9322e".DigitalOutput04;
	Cyclic#1.egmio:EGMModule3Out[4] AT %QX."X20DO9322e".DigitalOutput05;
	Cyclic#1.egmio:EGMModule3Out[5] AT %QX."X20DO9322e".DigitalOutput06;
	Cyclic#1.egmio:EGMModule3Out[6] AT %QX."X20DO9322e".DigitalOutput07;
	Cyclic#1.egmio:EGMModule3Out[7] AT %QX."X20DO9322e".DigitalOutput08;
	Cyclic#1.ModulStatus_DI AT %IX."X20DI9371b".ModuleOk;
	Cyclic#1.egmio:EGMModule1In[0] AT %IX."X20DI9371b".DigitalInput01;
	Cyclic#1.egmio:EGMModule1In[1] AT %IX."X20DI9371b".DigitalInput02;
	Cyclic#1.egmio:EGMModule1In[2] AT %IX."X20DI9371b".DigitalInput03;
	Cyclic#1.egmio:EGMModule1In[3] AT %IX."X20DI9371b".DigitalInput04;
	Cyclic#1.egmio:EGMModule1In[4] AT %IX."X20DI9371b".DigitalInput05;
	Cyclic#1.egmio:EGMModule1In[5] AT %IX."X20DI9371b".DigitalInput06;
	Cyclic#1.egmio:EGMModule1In[6] AT %IX."X20DI9371b".DigitalInput07;
	Cyclic#1.egmio:EGMModule1In[7] AT %IX."X20DI9371b".DigitalInput08;
	Cyclic#1.egmio:EGMModule1In[8] AT %IX."X20DI9371b".DigitalInput09;
	Cyclic#1.egmio:EGMModule1In[9] AT %IX."X20DI9371b".DigitalInput10;
	Cyclic#1.ModulStatus_AT AT %IX."X20AT4222".ModuleOk;
	Cyclic#1.EGMPreheat.AmbientTemp[0] AT %IW."X20AT4222".Temperature01;
	Cyclic#1.devtank:TempSensorValue AT %IW."X20AT4222".Temperature02;
	Cyclic#1.ModulStatus_AT1 AT %IB."X20AT4222".StatusInput01;
	ModulStatus_AO AT %IX."X20AO2622".ModuleOk;
	Cyclic#1.EGMMainMotor.RatedRpm AT %QW."X20AO2622".AnalogOutput01;
	Cyclic#1.EGMBrushMotor.RatedRpm AT %QW."X20AO2622".AnalogOutput02;
	Cyclic#1.ModulStatus_PS AT %IX."X20PS9400a".ModuleOk;
	Cyclic#1.ModulStatus_PS1 AT %IX."X20PS9400a".StatusInput01;
	Cyclic#1.ModulStatus_PS2 AT %IX."X20PS9400a".StatusInput02;
	Cyclic#1.ModulStatus_DI2 AT %IX."X20DI9371c".ModuleOk;
	Cyclic#1.egmio:EGMModule2In[0] AT %IX."X20DI9371c".DigitalInput01;
	Cyclic#1.egmio:EGMModule2In[1] AT %IX."X20DI9371c".DigitalInput02;
	Cyclic#1.egmio:EGMModule2In[2] AT %IX."X20DI9371c".DigitalInput03;
	Cyclic#1.egmio:EGMModule2In[3] AT %IX."X20DI9371c".DigitalInput04;
	Cyclic#1.egmio:EGMModule2In[4] AT %IX."X20DI9371c".DigitalInput05;
	Cyclic#1.egmio:EGMModule2In[5] AT %IX."X20DI9371c".DigitalInput06;
	Cyclic#1.EGMPreheat.RealTemp[0] AT %IW."X20AT4222".Temperature03;
	Cyclic#1.EGMPreheat.RealTemp[1] AT %IW."X20AT4222".Temperature04;
	Cyclic#1.egmio:EGMModule1In[10] AT %IX."X20DI9371b".DigitalInput11;
	Cyclic#1.egmio:EGMModule2Out[7] AT %QX."X20DO9322d".DigitalOutput08;
	Cyclic#1.egmio:EGMModule2Out[8] AT %QX."X20DO9322d".DigitalOutput09;
	Cyclic#1.egmio:EGMModule2Out[9] AT %QX."X20DO9322d".DigitalOutput10;
	Cyclic#1.egmio:EGMModule2Out[10] AT %QX."X20DO9322d".DigitalOutput11;
	Cyclic#1.egmio:EGMModule2Out[11] AT %QX."X20DO9322d".DigitalOutput12;
	Cyclic#1.egmio:EGMModule3Out[8] AT %QX."X20DO9322e".DigitalOutput09;
	Cyclic#1.egmio:EGMModule3Out[9] AT %QX."X20DO9322e".DigitalOutput10;
	Cyclic#1.egmio:EGMModule3Out[10] AT %QX."X20DO9322e".DigitalOutput11;
	Cyclic#1.egmio:EGMModule3Out[11] AT %QX."X20DO9322e".DigitalOutput12;
	Cyclic#1.egmio:EGMModule1In[11] AT %IX."X20DI9371b".DigitalInput12;
	Cyclic#1.egmio:EGMModule2In[6] AT %IX."X20DI9371c".DigitalInput07;
	Cyclic#1.egmio:EGMModule2In[7] AT %IX."X20DI9371c".DigitalInput08;
	Cyclic#1.egmio:EGMModule2In[8] AT %IX."X20DI9371c".DigitalInput09;
	Cyclic#1.egmio:EGMModule2In[9] AT %IX."X20DI9371c".DigitalInput10;
	Cyclic#1.egmio:EGMModule2In[10] AT %IX."X20DI9371c".DigitalInput11;
	Cyclic#1.egmio:EGMModule2In[11] AT %IX."X20DI9371c".DigitalInput12;
	Cyclic#1.In_ServiceMode AT %IX."X20DI9371".DigitalInput01;
	Cyclic#1.In_PaperSensor[0] AT %IX."X20DI9371".DigitalInput03;
	Cyclic#1.In_PaperSensor[1] AT %IX."X20DI9371".DigitalInput04;
	Cyclic#1.In_FeederHorActive AT %IX."X20DI9371".DigitalInput05;
	Cyclic#1.In_FeederHorInactive AT %IX."X20DI9371".DigitalInput06;
	Cyclic#1.In_FeederVacuumOK[0] AT %IX."X20DI9371".DigitalInput07;
	Cyclic#1.In_FeederVacuumOK[1] AT %IX."X20DI9371".DigitalInput08;
	Cyclic#1.In_FeederVacuumOK[2] AT %IX."X20DI9371".DigitalInput09;
	Cyclic#1.In_FeederVacuumOK[3] AT %IX."X20DI9371".DigitalInput10;
	Cyclic#1.In_FeederVacuumOK[4] AT %IX."X20DI9371".DigitalInput11;
	Cyclic#1.In_FeederVacuumOK[5] AT %IX."X20DI9371".DigitalInput12;
	Cyclic#1.In_PlateAdjusted[0] AT %IX."X20DI9371a".DigitalInput01;
	Cyclic#1.In_PlateAdjusted[1] AT %IX."X20DI9371a".DigitalInput02;
	Cyclic#1.In_LiftingPinsDown AT %IX."X20DI9371a".DigitalInput03;
	Cyclic#1.In_ConveyorBeltSensor[0] AT %IX."X20DI9371a".DigitalInput04 INVERSE;
	Cyclic#1.In_ConveyorBeltSensor[1] AT %IX."X20DI9371a".DigitalInput05 INVERSE;
	Cyclic#1.TrolleyCodeSensor AT %IX."X20DI9371a".DigitalInput07;
	Cyclic#1.BeltLoose AT %IX."X20DI9371a".DigitalInput08;
	Cyclic#1.in_out:Module4[0] AT %QX."X20DO9322".DigitalOutput01;
	Cyclic#1.in_out:Module4[1] AT %QX."X20DO9322".DigitalOutput02;
	Cyclic#1.in_out:Module4[2] AT %QX."X20DO9322".DigitalOutput03;
	Cyclic#1.in_out:Module4[3] AT %QX."X20DO9322".DigitalOutput04;
	Cyclic#1.in_out:Module4[4] AT %QX."X20DO9322".DigitalOutput05;
	Cyclic#1.in_out:Module4[5] AT %QX."X20DO9322".DigitalOutput06;
	Cyclic#1.in_out:Module4[6] AT %QX."X20DO9322".DigitalOutput07;
	Cyclic#1.in_out:Module4[7] AT %QX."X20DO9322".DigitalOutput08;
	Cyclic#1.in_out:Module4[8] AT %QX."X20DO9322".DigitalOutput09;
	Cyclic#1.in_out:Module4[9] AT %QX."X20DO9322".DigitalOutput10;
	Cyclic#1.in_out:Module4[10] AT %QX."X20DO9322".DigitalOutput11;
	Cyclic#1.in_out:Module4[11] AT %QX."X20DO9322".DigitalOutput12;
	Cyclic#1.in_out:Module5[0] AT %QX."X20DO9322a".DigitalOutput01;
	Cyclic#1.in_out:Module5[1] AT %QX."X20DO9322a".DigitalOutput02;
	Cyclic#1.in_out:Module5[2] AT %QX."X20DO9322a".DigitalOutput03;
	Cyclic#1.in_out:Module5[3] AT %QX."X20DO9322a".DigitalOutput04;
	Cyclic#1.in_out:Module5[4] AT %QX."X20DO9322a".DigitalOutput05;
	Cyclic#1.in_out:Module5[5] AT %QX."X20DO9322a".DigitalOutput06;
	Cyclic#1.in_out:Module5[6] AT %QX."X20DO9322a".DigitalOutput07;
	Cyclic#1.in_out:Module5[7] AT %QX."X20DO9322a".DigitalOutput08;
	Cyclic#1.in_out:Module5[8] AT %QX."X20DO9322a".DigitalOutput09;
	Cyclic#1.in_out:Module5[9] AT %QX."X20DO9322a".DigitalOutput10;
	Cyclic#1.in_out:Module5[10] AT %QX."X20DO9322a".DigitalOutput11;
	Cyclic#1.in_out:Module5[11] AT %QX."X20DO9322a".DigitalOutput12;
	Cyclic#1.in_out:Module6[0] AT %QX."X20DO9322b".DigitalOutput01;
	Cyclic#1.in_out:Module6[1] AT %QX."X20DO9322b".DigitalOutput02;
	Cyclic#1.in_out:Module6[2] AT %QX."X20DO9322b".DigitalOutput03;
	Cyclic#1.in_out:Module6[3] AT %QX."X20DO9322b".DigitalOutput04;
	Cyclic#1.in_out:Module6[4] AT %QX."X20DO9322b".DigitalOutput05;
	Cyclic#1.in_out:Module6[5] AT %QX."X20DO9322b".DigitalOutput06;
	Cyclic#1.in_out:Module6[6] AT %QX."X20DO9322b".DigitalOutput07;
	Cyclic#1.in_out:Module6[7] AT %QX."X20DO9322b".DigitalOutput08;
	Cyclic#1.in_out:Module6[8] AT %QX."X20DO9322b".DigitalOutput09;
	Cyclic#1.in_out:Module6[9] AT %QX."X20DO9322b".DigitalOutput10;
	Cyclic#1.in_out:Module6[10] AT %QX."X20DO9322b".DigitalOutput11;
	Cyclic#1.in_out:Module6[11] AT %QX."X20DO9322b".DigitalOutput12;
	Cyclic#1.CoverLockOK AT %IX."X20DI9371a".DigitalInput09;
	Cyclic#1.DoorsOK AT %IX."X20DI9371a".DigitalInput10;
	Cyclic#1.::CPUTemp AT %IW."5PPC2100_BY01_000".TemperatureCPU;
	Cyclic#1.::AmbientTemp AT %IW."5PPC2100_BY01_000".TemperatureRAM;
END_VAR
```

## Logical view

Binary libraries used (declarations not repeated): visapi, sys_lib, runtime, standard, operator, LoopCont 3.01.0, brsystem, inaclnt, FileIO, ETHSOCK, ETHERNET, dvframe, DataObj, Convert, CAN_Lib, AsUDP, astime, asstring, AsIOMMan, AsIMA, AsARCfg

### auxfunc.h
```c
/*
                             *******************
******************************* C HEADER FILE *******************************
**                           *******************                           **
**                                                                         **
** project  : LS JET II                                                    **
** filename : AUXFUNC.H                                                    **
** version  : 1.00                                                         **
** date     : 27.10.2006                                                   **
**                                                                         **
*****************************************************************************
** Abstract                                                                **
** ========                                                                **
** Declares the functions for common features          	                   **
**                                                                         **
**                                                                         **
** Copyright (c) 2006, Krause-Biagosch GmbH                                **
** All rights reserved.                                                    **
**                                                                         **
*****************************************************************************
VERSION HISTORY:
----------------
Version     : 1.00
Date        : 27.10.2006
Revised by  : Herbert Aden
Description : Original version.
*/

#ifndef _AUXFUNC_INCLUDED
#define _AUXFUNC_INCLUDED

/****************************************************************************/
/**                                                                        **/
/**                           INCLUDE FILES                                **/
/**                                                                        **/
/****************************************************************************/
#include "glob_var.h"

/****************************************************************************/
/**                                                                        **/
/**                       DEFINITIONS AND MACROS                           **/
/**                                                                        **/
/****************************************************************************/
/* NONE */

/****************************************************************************/
/**                                                                        **/
/**                      TYPEDEFS AND STRUCTURES                           **/
/**                                                                        **/
/****************************************************************************/
#undef CAUTION
#undef INFO
#undef REQUEST
enum IconType   {CAUTION, INFO, REQUEST};
enum ButtonType {NONE, OKONLY, OKCANCEL};

/****************************************************************************/
/**                                                                        **/
/**                      EXPORTED VARIABLES                                **/
/**                                                                        **/
/****************************************************************************/
#ifndef _AUXFUNC_C_SRC
#endif

/****************************************************************************/
/**                                                                        **/
/**                          EXPORTED FUNCTIONS                            **/
/**                                                                        **/
/****************************************************************************/

void ShowMessage(const int T1,const int T2,const int T3,
                 const int Icon, const int Button, const BOOL pIgnoreButtons);

void SwitchFeederVacuum(USINT PlateType, USINT Config, BOOL fct);
void SwitchAdjustVacuum(USINT PlateType, USINT Config, BOOL fct);
void SwitchAdjustTableVacuum(USINT PlateType, USINT Config, BOOL fct);
BOOL CheckFeederVacuum(USINT PlateType, USINT Config);
BOOL CheckAdjustVacuum(USINT PlateType, USINT Config);
BOOL CheckForPaper(USINT Config);
void MoveAdjustSucker(USINT Config, USINT fct);
BOOL AdjustOK(USINT Config);
BOOL AdjPins(USINT Config,USINT *Step, TON_10ms_typ *Timer);
void ClearStation(PlateInSystem_Type *Station);

#endif
/****************************************************************************/
/**                                                                        **/
/**                                 EOF                                    **/
/**                                                                        **/
/****************************************************************************/
```

### bit_func.h
```c
/****************************************************************************/
/*	Headermodul für Bitbehandlungsfunktionen								*/
/*																			*/
/*	Änderungsdatum:		15.03.00											*/
/*																			*/
/****************************************************************************/

#define BIT_SET(x,y) ( x | (1 << y))
#define BIT_CLR(x,y) ( x & ~(1 << y))
#define BIT_TST(x,y) ( (x & (1 << y)) != 0 ? 1 : 0)
#define NOT(x)		 (x == 0 ? 1 : 0)
```

### egmglob_var.h
```c
/*************************************************************************************************
 Global header file for EGM

 defines, global variables and common includes

*************************************************************************************************/

#include <bur/plc.h>       /* macros for B&R PLC programming */
#include <bur/plctypes.h>
#include <standard.h>      /* prototypes for STANDARD-Library */
#include <sys_lib.h>
#include <asstring.h>
#include <string.h>
#include <loopcont.h>

#ifndef TRUE
	#define  TRUE (1)
#endif
#ifndef FALSE
	#define FALSE (0)
#endif
#define MAXPLATETYPES (10)
#define MAXPLATETYPENAME 20
/*Modes*/
#define M_OFF 0
#define M_AUTO 1
#define M_INITCLEANING 2
#define M_CLEANING 3

/*States*/
#define S_OFF 0
#define S_HEATING 1
#define S_READY 2
#define S_STARTPROCESSING 3
#define S_PROCESSING 4
#define S_WAITFORSTANDBY 5
#define S_CLEANING1 6
#define S_CLEANING2 7
#define S_CLEANING3 8
#define S_ERROR 10

#define CAUTION 0
#define INFO	1
#define REQUEST	2

#define MESSAGEPIC 41
#define FILEPIC 42
#define EMPTYPIC 107

#define	MAXFILELIST	32
#define MAXFILES	50
#define MAXFILENAMELENGTH	32

#define EGMSRAMSIZEWORDS 2500
#define EGMSRAMSIZEBYTES 5000

#define OVERALLSRAMSIZEWORDS 12500
#define OVERALLSRAMSIZEEBYTES 25000

#define PERFSRAMSIZEWORDS 10000
#define PERFSRAMSIZEBYTES 20000

#define OPEN		(1)
#define CLOSE	(0)
#ifndef ON
	#define ON		(1)
#endif
#ifndef OFF
	#define OFF		(0)
#endif

#define REPLPERSQM (1)
#define REPLPERPLATE (2)
#define FRESHWATERONLY (3)

#define FIFOLENGTH		(10)

#define EGM_MAXALARMS	(99)

enum PlateState {PS_NONE=0, PS_RUNNING, PS_WAITINGFOROUTPUT, PS_OUTPUTREACHED};

#define MAX_NUMBER_OF_CONTROLLERS	4

#define BLUEFIN_XS (1)
#define BLUEFIN_LOWCHEM (2)

/***************************** Type Definitions ***********************************/
typedef struct
{
	CTUtyp	EdgeCounter;
	INT		LastCV;
	INT		Frequency;
	INT		FlowCounter;
	INT		OverflowCounter;
	REAL	LitersPerHour;
	REAL	LitersPerMinute;
	DINT	MlFlown;
	BOOL	ResetMlFlown;
	BOOL	Flowing;
	UDINT	PulsesPerLiter;
}FlowCount_type;

typedef struct
{
	STRING Name[MAXPLATETYPENAME];
	STRING ManufacturerName[20];
	UDINT	SizeX;
	UDINT	SizeY;
/* Fläche der Platte (ergibt sich natürlich aus SizeX*SizeY */
	REAL	Area;
/* Regeneratverbrauch pro Quadratmeter */
	REAL	RegenerationPerSqrM;
/* Regeneratverbrauch pro Platte */
	REAL	RegenerationPerPlate;
/* Plattentyp (Silber, Polymer oder was immer */
	USINT	Type;
/*Dip Zeit in s*/
	USINT	DipTime;
/*20 Bytes reserve*/
	UDINT Reserve[5];
} EGMPlate_Type;

/***********************************************************/
/* Developer */
typedef struct
{
	STRING	Name[20];
	UINT		Temperature;				/* 0,1 °C*/
	UINT		Lifetime;					/* Days */
	UINT		MaxArea;					/* m² */
	UINT		TopUp;					/* ml/m² */
	REAL		Replenishment;			/* ml/m² */
	REAL		StandbyReplenishment;	/* ml/h */
	UINT		BrushSpeed;				/* rpm (mit Faktor für Visualisierung!)*/
} EGMDeveloper_Type;

typedef struct
{
	STRING Version[10];
	USINT MachineType;
	USINT	Unit_Rpm; /*rpm oder Hz*/
	USINT	Unit_Propulsion; /*m/min oder ft/min*/
	USINT	Unit_Temperature; /*C oder F*/
	USINT	Unit_Length; /*mm oder Inch*/
	USINT	Unit_Area; /*quadratmeter oder squareInch*/
	USINT	Unit_Volume; /* Liter oder Gallone*/
/*Factor Rpm<->PlateSpeed in m/min*/
	REAL	MainMotorFactor;
	REAL	CurrentPlateSpeed; /*m/min*/
	UDINT	CurrentDipTime; /*s*/
	UDINT	CurrentBrushSpeed; /*rpm*/
	UDINT	MaxPlateSizeX;
	UDINT	MaxPlateSizeY;
/* added 18.01.2007*/
	REAL	BrushFactor;
	STRING	MachineNumber[10];
/* Flow control einzeln aktivierbar */
	BOOL	UseGumFlowControl;
	BOOL	UseDevCircFlowControl;
	BOOL	UsePrewashFlowControl;
	BOOL	UseRinseFlowControl;
	BOOL	UseTopUpFlowControl;
	BOOL	UseReplFlowControl;
	BOOL	PlateDirection;	/* 0=right to left, 1=left to right */
	USINT	PROV_KitInstalled;	/* */
	BOOL	CheckIfCoolingDeviceOk;
	UDINT	DeveloperPulsesPerLiter;
	UDINT	ReplenisherPulsesPerLiter;
	UDINT	GumPulsesPerLiter;
	UDINT	ScreensaverTime; /* in sec */
	BOOL	EnableGumSection; /* neu für LowChem: Gummierung ist optional bei LC*/
} EGMGlobalParam_Type;

/* Motors */

typedef struct
{
	BOOL	Enable;	/*Freigabe Ausgang (EIN)*/
	USINT	Auto;
	USINT	Manual;
	USINT	Start;
	USINT	Stop;
	INT	RatedRpm; /*in cm/min wg Genauigkeit*/
	INT		AutoRatedRpm;
	INT		RealRpm;
/*20 Bytes reserve*/
	UDINT Reserve[5];
} EGMMotor_Type;

typedef struct
{
	REAL	Kp;
	REAL	Tn;
	REAL	Tv;
	REAL	Tf;
	REAL	Kw;
	REAL	Kfbk;
	USINT	d_mode;
	UINT	tminpuls;
	UINT	tperiod;
	BOOL	SetpointTracking;
}EGMReglerParam_typ;

typedef struct
{
	UINT	RatedTemp[4];
/*Bereich, der als OK betrachtet wird*/
	UINT	ToleratedDevPos;
	UINT	ToleratedDevNeg;

	UINT	MaxOKTemp; /*ergeben sich automatisch aus ToleratedDev...*/
	UINT	MinOKTemp; /*ergeben sich automatisch aus ToleratedDev...*/

	INT		RatedTempCorr[4];
	EGMReglerParam_typ		ReglerParam[4];
	UINT	SetPointCorrTMin;	/*Sollwertnachf. Zeitkonst in Min*/
	UINT	SetPointCorrMax;		/*Sollwertnachf. Maxwert in °C*/
/*Wertepaare für Korrekturgeraden*/
	UINT	EndSetpoint[5];
	UINT	StartOverheat[5];
	UINT	StartAmbient[5];
	UINT	EndAmbient[5];

	INT		DecPerPlate;
	INT		IncPerMinute;
	INT		MaxInc;
	INT		AmbientThreshold;
} EGMPreheatParam_Type;

typedef struct
{
	BOOL	Enable;
	BOOL	Auto[4];

/*
4 Heizkreise vorgesehen
bisher [0] und [1] verwendet,
[2] nichtz benutzt
[3] für Umgebungstemperatur
*/
	INT RealTemp[4];
/* Umgebungstemp (4 mal vorgesehen als Reserve) */
	INT AmbientTemp[4];
/*4 Heizkreise vorgesehen*/
	INT		HeatingOn[4];

/*Ausgang: Bereit, Temp OK*/
	USINT	TempInRange;
	USINT	TempNotInRange;
/* Schaltausgang Lüfter */
	BOOL	FansOn;

} EGMPreheat_Type;

typedef struct
{
	UDINT	RatedTemp;

/*Bereich, der als OK betrachtet wird*/
	UINT	ToleratedDevPos;
	UINT	ToleratedDevNeg;

/*Hysterese f Heizung*/
/**/
	UINT	SwitchDevHeatingOn;
	UINT	SwitchDevHeatingOff;
	UINT	SwitchDevCoolingOn;
	UINT	SwitchDevCoolingOff;

	UINT	HeatingOnTemp; /*ergeben sich automatisch aus Switchdev...*/
	UINT	HeatingOffTemp; /*ergeben sich automatisch aus Switchdev...*/
/*Kühlung Einschaltpunkt*/
	INT		CoolingOnY;
/*Kühlung Ausschaltpunkt*/
	UINT	CoolingOffTemp;

	UINT	MaxOKTemp; /*ergeben sich automatisch aus ToleratedDev...*/
	UINT	MinOKTemp; /*ergeben sich automatisch aus ToleratedDev...*/

/*Wartezeiten, um stabile Zustände abzuwarten (im Prinzip der I-Anteil)*/
	UINT	HeatingOnDelay;
	UINT	HeatingOffDelay;
	UINT	CoolingOnDelay;
	UINT	CoolingOffDelay;
/*min/max Ein/Ausschaltzeiten*/
	UINT	MaxOnTimeHeating;
	UINT	MinOnTimeHeating;
	UINT	MaxOffTimeHeating;
	UINT	MinOffTimeHeating;
	UINT	MaxOnTimeCooling;
	UINT	MinOnTimeCooling;
	UINT	MaxOffTimeCooling;
	UINT	MinOffTimeCooling;

	UDINT	StartRefillDelay; /*s*/
	UDINT	StopRefillDelay; /*s*/
	EGMReglerParam_typ		ReglerParam;
/* Replenishing*/
	UINT	DeveloperType; /*Nummer des Entwicklers aus Liste*/
	STRING	DeveloperName[20];
	UINT		ReplenishingMode;	/* per m², per plate */
	BOOL		EnableStandbyReplenishing;
	BOOL		EnableOffReplenishing;
	UINT		TopUpMode;	/* per m², per plate */
	REAL		ReplenishmentPerSqm;	/* ml/m² */
	REAL		ReplenishmentPerPlate;	/* ml/pl */
	REAL		StandbyReplenishment;	/* ml/h */
	REAL		OffReplenishment;	/* ml/h */
	UINT		StandbyReplenishmentIntervall;	/* min */
	REAL		PumpMlPerSec;			/* ml/s */
	UINT		MinPumpOnTime;			/* 10 ms */
	UINT		MinPumpOnTimeStandby;			/* 10 ms */
	INT			TempOffset;
	REAL		TopUpPerSqm;	/* ml/m² */
	REAL		TopUpPerPlate;	/* ml/pl */
	REAL		TopUpPumpMlPerSec;			/* ml/s */
	UINT		TopUpMinPumpOnTime;			/* 10 ms */
} EGMDeveloperTankParam_Type;

typedef struct
{
	BOOL	Enable;
	BOOL	Auto;
	INT		RealTemp;
/*in/out*/
	BOOL	TankFull;
	BOOL	TankEmpty;
	BOOL	RegenerationPump;
	BOOL	CirculationPump;
	BOOL	Refill;
	BOOL	HeatingOn;
	BOOL	CoolingOn;

/*Ausgang: Bereit, Temp OK*/
	USINT	TempInRange;
	USINT	TempNotInRange;

	USINT	LevelInRange;
	USINT	LevelNotInRange;
} EGMDeveloperTank_Type;

typedef struct
{
	UINT	Speed;
	UINT	BrushSpeed;
	UINT	PreheatTemp;
	UINT	DeveloperTemp;
	UINT	StandbyDelay;
	UINT	StandbySpeed;
	REAL	MaxPlateSizeX;
	REAL	MaxPlateSizeY;
	UINT	StandbyBrushSpeed;
	UINT	PreheatTemp2;
/*die nächsten 3 Zeiten in sec*/
	UINT	WaitGumBackTime;
	UINT	GumRinsingTime;
	UINT	WaitGumRinseTime;
/* PRO V Erweiterungen */
	UINT	PROV_PumpOnTime;
	UINT	PROV_PumpOffTime;
} EGMAutoParam_Type;

typedef struct
{
/*IN / OUT*/
	BOOL	TankFull;
	BOOL	Pump;
	BOOL	Valve;
	BOOL	HeatingOn;
	USINT		LevelNotInRange;
	INT		RealTemperature;
	BOOL	Auto;
	BOOL	PumpCmd;
} EGMPrewash_Type;

typedef struct
{
	UINT		ReplenishingMode;	/* per m², per plate, freshwater only */
	REAL		ReplenishmentPerSqm;	/* ml/m² */
	REAL		ReplenishmentPerPlate;	/* ml/pl */
	UINT		ReplenishmentIntervall;	/* min */
	REAL		PumpMlPerSec;			/* ml/s */
	UINT		MinPumpOnTime;			/* 10 ms */

} EGMPrewashParam_Type;

typedef struct
{
	UINT		ReplenishingMode;	/* per m², per plate */
	REAL		ReplenishmentPerSqm;	/* ml/m² */
	REAL		ReplenishmentPerPlate;	/* ml/pl */
	UINT		ReplenishmentIntervall;	/* min */
	REAL		PumpMlPerSec;			/* ml/s */
	UINT		MinPumpOnTime;			/* 10 ms */

} EGMRinseParam_Type;

typedef struct
{
/*IN / OUT*/
	BOOL	TankFull;
	BOOL	Pump;
	BOOL	Valve;
	USINT		LevelNotInRange;
	BOOL	Auto;
	BOOL	PumpCmd;

} EGMRinse_Type;

typedef struct
{
/*IN / OUT*/
	BOOL	TankFull;
	BOOL	Pump;
	BOOL	Valve;			/* Umschalten: 0->Ablauf in Abfluß, 1->Ablauf in Gummierungsbehälter*/
	BOOL	RinseValve;	/* Spülwasser */
	USINT		LevelNotInRange;
	BOOL	Auto;
	BOOL	PumpCmd;
} EGMGum_Type;

typedef struct
{
	BOOL	Used;
	UINT	Type;
	REAL	Position;
	REAL	Length;
	USINT	Status;
}EGMPlate_FIFO_Type;

typedef struct
{
	UINT	mode;
	UINT	state;
	UINT	ErrorNumber;
	STRING	ErrorText[64];
}EGMState_struct;

typedef struct
{
	REAL	SetPoint;
	REAL	LimitLow;
	REAL	LimitHigh;
	REAL	HeatP;
	REAL	HeatI;
	REAL	HeatD;
	REAL	CoolP;
	REAL	CoolI;
	REAL	CoolD;

}Cooler_Values;

typedef struct
{
	USINT	RawDataB1;
	USINT	RawDataB2;
	USINT	RawDataB3;
	USINT	RawDataB4;
	USINT	RawDataB5;

	BOOL	RTD1OpenFault;
	BOOL	RTD1ShortedFault;
	BOOL	RTD1Open;
	BOOL	RTD1Shorted;
	BOOL	RTD2OpenFault;
	BOOL	RTD2ShortedFault;
	BOOL	RTD2Open;
	BOOL	RTD2Shorted;
	BOOL	RTD2OpenWarn;
	BOOL	RTD2ShortedWarn;
	BOOL	RTD3OpenFault;
	BOOL	RTD3ShortedFault;
	BOOL	RTD3Open;
	BOOL	RTD3Shorted;
	BOOL	RefrigHighTemp;
	BOOL	HTCFault;
	BOOL	HighFixedTempFault;
	BOOL	LowFixedTempFault;
	BOOL	HighTempFault;
	BOOL	LowTempFault;
	BOOL	LowLevelFault;
	BOOL	HighTempWarn;
	BOOL	LowTempWarn;
	BOOL	LowLevelWarn;
	BOOL	BuzzerOn;
	BOOL	AlarmMuted;
	BOOL	UnitFaulted;
	BOOL	UnitStopping;
	BOOL	UnitOn;
	BOOL	PumpOn;
	BOOL	CompressorOn;
	BOOL	HeaterOn;
	BOOL	RTD2Controlling;
	BOOL	HeatLEDFlashing;
	BOOL	CoolLEDFlashing;
	BOOL	CoolLEDOn;

	BOOL	Cmd_Start;
	BOOL	Cmd_Stop;

	Cooler_Values CurrentValues;
	Cooler_Values NewValues;

	REAL	IntTemp;
	REAL	ExtTemp;

} Cooler_struct;

/***************************** Variable Definitions ***********************************/

_GLOBAL STRING  EGMgVERSION[9];

_GLOBAL USINT UserLevel;
_GLOBAL USINT Language;
_GLOBAL USINT CurrentMode;
_GLOBAL USINT CurrentState;

_GLOBAL	EGMMotor_Type	EGMBrushMotor;
_GLOBAL	EGMMotor_Type	EGMMainMotor;
_GLOBAL	EGMAutoParam_Type		EGMAutoParam;

_GLOBAL	EGMDeveloperTank_Type	EGMDeveloperTank;
_GLOBAL	EGMPreheat_Type	EGMPreheat;
_GLOBAL	EGMPrewash_Type	EGMPrewash;
_GLOBAL	EGMRinse_Type	EGMRinse;
_GLOBAL	EGMGum_Type	EGMGum;

_GLOBAL	EGMPreheatParam_Type		EGMPreheatParam;
_GLOBAL	EGMGlobalParam_Type		EGMGlobalParam;
_GLOBAL	EGMDeveloperTankParam_Type		EGMDeveloperTankParam;
_GLOBAL	EGMPrewashParam_Type	EGMPrewashParam;
_GLOBAL	EGMRinseParam_Type	EGMRinseParam;

/* GENERAL INPUTS*/
_GLOBAL	BOOL	ControlVoltageOk;
_GLOBAL	BOOL	RPMCheck;
_GLOBAL 	BOOL	InputSensor;
_GLOBAL	BOOL	OutputSensor;

_GLOBAL BOOL		GumFlowInput;
_GLOBAL BOOL		ReplFlowInput;
_GLOBAL BOOL		TopUpFlowInput;
_GLOBAL BOOL		DevCircFlowInput;
_GLOBAL BOOL		PrewashFlowInput;
_GLOBAL BOOL		RinseFlowInput;
_GLOBAL	BOOL		ServiceKey;
_GLOBAL	BOOL		PlateSensor;
_GLOBAL	BOOL		VCP_OK;

/* GENERAL OUTPUTS*/
_GLOBAL	BOOL	Ready;
_GLOBAL	BOOL	NoError;
_GLOBAL	BOOL	ActivateControlVoltage;
_GLOBAL	BOOL	Drying;
_GLOBAL	BOOL	LightGreen;
_GLOBAL	BOOL	LightYellow;
_GLOBAL	BOOL	LightRed;
_GLOBAL	BOOL	Horn;

/*Zeitbasiswerte für Regelung*/
_GLOBAL	LCCounter_typ LCCountVar;

/*Plattentypen*/
_GLOBAL	EGMPlate_Type EGMPlateTypes[MAXPLATETYPES];

/* Var für Darstellung der Platten auf dem Schirm*/
_GLOBAL	EGMPlate_FIFO_Type	EGMPlateFIFO[FIFOLENGTH];
_GLOBAL	UINT	EGMPlatesInFIFO;

/* Var for replenishment managament. used in Developertank task*/
_GLOBAL UINT	ReplenishmentPlateCounter,PrewashReplenishmentPlateCounter,
					RinseReplenishmentPlateCounter,TopUpPlateCounter;
_GLOBAL REAL	ReplenishmentSqmCounter,PrewashReplenishmentSqmCounter,
					RinseReplenishmentSqmCounter,TopUpSqmCounter;

_GLOBAL UDINT	OverallPlateCounter _VAR_RETAIN,OverallReplenisherCounter _VAR_RETAIN,ReplenisherCounter	_VAR_RETAIN,
OverallReplenisherPumpTime _VAR_RETAIN;
_GLOBAL REAL		OverallSqmCounter	_VAR_RETAIN;

_GLOBAL UINT	SessionPlateCounter;
_GLOBAL REAL	SessionSqmCounter;
_GLOBAL REAL	SqmSinceDevChg	_VAR_RETAIN;
_GLOBAL UDINT	ReplenisherUsedSinceDevChg	_VAR_RETAIN;
_GLOBAL	UDINT	DeveloperChangeDate _VAR_RETAIN,ReplenisherUsedSinceDevChange	_VAR_RETAIN;

_GLOBAL	BOOL	EGM_AlarmBitField[EGM_MAXALARMS],EGM_AlarmQuitBitField[EGM_MAXALARMS];
_GLOBAL	UINT	CPUTemp,AmbientTemp;
_GLOBAL	USINT	BatteryStatus;
_GLOBAL	EGMState_struct	EGMState;
_GLOBAL	Cooler_struct Cooler;
_GLOBAL	BOOL	ModulStatus_DO1,ModulStatus_DO2,ModulStatus_DO3,
ModulStatus_DI,ModulStatus_DI2,ModulStatus_AT,
ModulStatus_AO,ModulStatus_PS,ModulStatus_PS1,ModulStatus_PS2;
_GLOBAL USINT	ModulStatus_AT1;
_GLOBAL	FlowCount_type	GumFC, ReplFC, TopUpFC;
_GLOBAL BOOL	HeatingON[MAX_NUMBER_OF_CONTROLLERS];
/* E/A für ProV Test Japan */
_GLOBAL	BOOL In_DevCanister_Full;
_GLOBAL	BOOL In_DevCanister_Empty;
_GLOBAL	BOOL Out_DevCanister_Circulation;
_GLOBAL	BOOL Out_DevCanister_Replenish;
/*
Maschinenlänge in m
	Standard Bluefin 2.80
	XS Bluefin		 2.70
	LowChem Bluefin  2.05
 */
_GLOBAL REAL MACHINELENGTH;
_GLOBAL USINT MachineType;
```

### glob_var.h
```c
/****************************************************************************/
/*	Globale Definitionen													*/
/*	Änderungsdatum:		13.08.01											*/
/*																			*/
/****************************************************************************/

#ifndef _GLOB_VAR_INCLUDED_
	#define _GLOB_VAR_INCLUDED_ 1

	/* INCLUDEs */
	#include	<bur/plctypes.h>
	#include 	<standard.h>

	/* !!! ACHTUNG!!  Bei Veränderungen in dieser Datei immer ALLES KOMPILIEREN !!!*/

	/*kennzeichnet die EasyLoad Version im Gegensatz zu LSJet*/
	#define PERFORMANCE

	/* Auswahl der Maschine: Performance, Bluefin oder Kombination*/

/*
	#define MODE_PERFORMANCE	0
	#undef MODE_BLUEFIN
	#undef MODE_BOTH
*/
	/*
	#define MODE_BLUEFIN	1
	#undef MODE_BOTH
	#undef MODE_PERFORMANCE
	*/

	/* Performance und Bluefin mit gemeinsamer Steuerung*/

	#define MODE_BOTH	2
	#undef MODE_BLUEFIN
	#undef MODE_PERFORMANCE

	/* defines */
	#define EIN			1
	#define AUS			0
#ifndef ON
	#define ON		(1)
#endif
#ifndef OFF
	#define OFF		(0)
#endif
#ifndef TRUE
	#define TRUE 		1
#endif
#ifndef FALSE
	#define FALSE 		0
#endif
	#define OK  		1
	#define NOT_OK 		0
	#define ACTIVE		1
	#define INACTIVE	0

	#define NOPLATE     99
	#define ALL	     	98
	#define	LEFT		0
	#define	RIGHT		1
	#define BOTH		2
	#define PANORAMA	3
	#define BROADSHEET	4
	#define PINS_DOWN	5

	#define	MAXALARMS	50

	#define MONOGON_MAX_SPEEDS 16
	#define WRITEDATALENGTH 20
	#define READDATALENGTH 60
	#define MAXMOTORS 20
	#define MAXTROLLEYS 10
	#define MAXPLATETYPES (10)
	#define MAXPLATETYPENAMELENGTH	32
	#define MAXTROLLEYNAMELENGTH	32
	#define MAXEXPOSEFILENAMELENGTH	128
	#define  JOBLISTSIZE			10
	#define  NO_JOB_RESERVED		(-1)
	#define  JOBIDLENGTH			(15)

	#define FEEDER_VERTICAL			1
	#define FEEDER_HORIZONTAL 		2
	#define SHUTTLE 				3
	#define PAPERREMOVE_HORIZONTAL 	4
	#define PAPERREMOVE_VERTICAL 	5
	#define ADJUSTER				6
	#define DELOADER_TURN			7
	#define DELOADER_HORIZONTAL		8
	#define CONVEYORBELT			9
	#define PAPERREMOVE_VERTICAL2 10

	#define CAUTION 0
	#define INFO	1
	#define REQUEST	2

	#define TABLELENGTH	1075
	#define MAXLASERPOWERSETTINGS 10
	#define TCPIPTIMEOUT 150

	#define MAXNUMBEROFTIFFBLASTERS (2)

	#define STREQ(a,b)    (strcmp ((a),(b))     == 0)
	#define STREQN(a,b,n) (strncmp((a),(b),(n)) == 0)

	#define S(a)	((SINT) (a))	     /* shortcut for cast to SINT (signed char)*/
	#define US(a)	((USINT) (a))	     /* shortcut for cast to USINT (unsigned char)*/
	#define I(a)	((INT) (a))	     /* shortcut for cast to INT (short int)*/
	#define UI(a)	((UINT) (a))	 /* shortcut for cast to UINT (unsigned short int)*/
	#define L(a)	((DINT) (a))	 /* shortcut for cast to DINT (signed long)*/
	#define UL(a)	((UDINT) (a))	 /* shortcut for cast to UDINT (unsigned long)*/

	#define SCREENSAVERPIC 5
	#define MESSAGEPIC 41
	#define FILEPIC 42

	#define MAXLASERPOWERSETTINGS 10

	#define NO_DELOADER               ((USINT) 0)
	#define DELOADER_ONLY             ((USINT) 1)
	#define DELOADER_AND_TURNSTATION  ((USINT) 2)

	#define NO_ROTATION	              ((USINT) 0)
	#define ROTATE_90                 ((USINT) 1)
	#define ROTATE_180                ((USINT) 2)

	/*--------------TYPES------------------------------------------------*/
	/* Datenstruktur Can Objekte*/
	typedef struct{
		unsigned char	InitRes[8];
		unsigned char	InitReq[8];
		unsigned char	StatRes[8];
		unsigned char	SteuReq[8];
		unsigned char	ParaRes[8];
		unsigned char	ParaReq[8];

		unsigned char	InitResEv;
		unsigned char	InitReqEv;
		unsigned char	StatResEv;
		unsigned char	SteuReqEv;
		unsigned char	ParaReqEv;
		unsigned char	ParaResEv;
	}CAN_OBJEKT_FUtyp;

	/* Datenstruktur für LUST CDD*/
	typedef struct
	{
	  unsigned char		SetPara;
	  unsigned char		GetPara;
	  unsigned short	IndexPara;
	  unsigned short	ParaStep;
	  unsigned short	IdxIntern;
	  unsigned char		Status;
	  unsigned char		DrvError[10];
	  unsigned short	timeoutCounter;
	  float				aktuellePosition_mm;/* aktuelle Position in mm*/
	  DINT				TargetPosition; 	/* Zielposition in Inkrementen*/
	  float				TargetPosition_mm; 	/*Eingegebene Zielposition (mm)*/
	  BOOL 				CANError;			/*Timeout oder CAN Komm Fehler*/
	/* vom Antrieb */
	  BOOL				Error;				/* allgemeiner Fehler */
	  BOOL				CANStatus;	 		/* 0=System Stop, 1=System Start */
	  BOOL				SollwertErreicht;
	  BOOL				Activ;				/* Endstufe aktiv */
	  BOOL				Rot0;				/* Drehzahl 0 */
	  BOOL				CReady;				/* Gerät betriebsbereit */
	  BOOL				ENPO;				/* ENPO Eingang */
	  BOOL				OSD00;				/* Ausgang OSD00 */
	  BOOL				OSD01;				/* Ausgang OSD01 */
	  BOOL				RefOk;				/* Referenzpunkt definiert */
	  BOOL				Auto;				/* Automatikbetrieb aktiv */
	  BOOL				Ablauf;				/* Ablaufprogramm aktiv */
	  BOOL				ZustandsMerker[8];	/* M80 bis M87 aus PosMod  */
	  BOOL				BefehlsMerker[8];	/* M90 bis M97 an PosMod  */
	  DINT				aktuellePosition;	/* aktuelle Position in Inkrementen*/
	/* Kommandos von Applikation */
	  BOOL				cmd_Start;			/* Regler Freigabe*/
	  BOOL				cmd_Auto;			/* Automatik/Handbetrieb*/
	  BOOL				cmd_tipp_plus;
	  BOOL				cmd_tipp_minus;
	  BOOL				cmd_tipp_schnell;
	  BOOL				cmd_Ref;
	  BOOL				cmd_Target;
	  BOOL				cmd_Park;
	  BOOL				cmd_Expose;
	/*interne Stati*/
	  BOOL				state_tipp_plus;
	  BOOL				state_tipp_minus;
	  BOOL				state_tipp_schnell;
	} FU_Typ;

	/* Datenstruktur für Parametrierung LUST CDD */
	typedef struct
	{
		UDINT ParaNr;
		UDINT Wert;
		USINT Index;
		BOOL Error;
		BOOL Ready;
	} FU_Para_Typ;

	/* Datenstruktur für Parameter X-Achse */
	typedef struct
	{
	/*Geschwindigkeiten*/
		UINT RefSpeed1;
		UINT RefSpeed2;
		UINT RefSpeed3;
		UINT ManSpeed1;
		UINT ManSpeed2;
		UINT ParkSpeed;
		REAL	MaxPosition;	/* Verfahrweg Ende plus*/
		REAL	MinPosition;	/* Verfahrweg Ende minus*/
	/*Positionen*/
		REAL Offset;		/*Nullpunktkorrektur*/
		REAL ParkPosition;
		REAL InkrementeProMm;
	} X_Param_Typ;				/* Länge: 24 Byte*/

	/* datenstruktur für Belichtungsparameter */
	typedef struct
	{
	/*Geschwindigkeiten*/
		REAL ExposeSpeed;		/* in mm/s */
		UINT MoveToStartSpeed; /* not yet used! controller uses ParkSpeed*/
	/*Positionen*/
		REAL StartPosition;		/* in mm */
		REAL PEGStartPosition;	/* in mm */
		REAL EndPosition;		/* in mm */
		REAL PEGEndPosition;	/* in mm */
		UINT Resolution;
		UDINT ScansPerMinute;
	} Expose_Param_Typ;

	/********************************************************************/
	/* Types for Faulhaber Motors	*/
	/********************************************************************/
	typedef struct
	{
		USINT	ControllerIFact;
		USINT 	Function[20];
		USINT	Priority;
		REAL	IncrementsPerMm;
		UDINT 	ReferenceSpeed;
		BOOL	ReferenceDirectionNegative;
		UDINT	ReferencePeekCurrent;
		UDINT	DefaultPeekCurrent;
		UDINT	ReferenceContCurrent;
		UDINT	DefaultContCurrent;
		UDINT	ReferencePropFact;
		UDINT	DefaultPropFact;
		UDINT	ReferenceOffset;
		UDINT	ReferenceAcceleration;
		UDINT	DefaultAcceleration;
		UDINT	ManSpeed;
		UDINT	MaximumSpeed;
		DINT	MaximumPosition;
		DINT	MinimumPosition;
		UDINT	PositionWindow;
	} Motor_Param_Typ;

	typedef struct
	{
		DINT 	Position;
		DINT 	LastPosition;
		REAL	Position_mm;
		BOOL	ReferenceOk;
		BOOL	Error;
		BOOL	Moving;
		BOOL	MovingPlus;
		BOOL	MovingMinus;
		USINT	ReferenceStep;
		USINT	timeout;
		BOOL	StartRef;
		Motor_Param_Typ	Parameter;
	}Motor_Typ;

	/* Datenstrukturen für Feeder */
	typedef struct
	{
		DINT		Up;
		DINT		AboveTrolley;
	/*V1.95 geänderte Funktion dieses Parameters: tiefste Position!*/
		DINT		MaxDown;
		DINT		PreRelease;
		DINT		ReleasePlate;
		DINT		EnablePaperRemove;
		DINT		SpeedChangePosition;  /* relative to platestack*/
	}Feeder_Vert_Pos_Typ;

	typedef struct
	{
		DINT		ReleasePlate;
		DINT		TakePlate;
	}Feeder_Horiz_Pos_Typ;

	typedef struct
	{
		UDINT		VacuumOnTime;		/* in 10ms */
		UDINT		VacuumOffTime;		/* in 10ms */
		UDINT		SpeedUpSlow;
		UDINT		SpeedUpFast;
		Feeder_Vert_Pos_Typ		VerticalPositions;
		Feeder_Horiz_Pos_Typ	HorizontalPositions;
		DINT		Stack0Pos;
		DINT		Stack20Pos;
		DINT		SlowDownPos;
		UDINT		StackDetectSpeed;
		DINT		PanoramaAdapter;
		USINT		SuckRepitions;
		USINT		ShakeRepitions;
		USINT		ShakeTime; /*in 10ms*/
		UDINT		ShakeWay;
		BOOL		WaitForExposer;		/*waiting on exposer start (avoid suction marks) on/off */
		BOOL		IgnoreVacuumSwitch;	/*don't check vacuum switch*/
		DINT		HorPositionPano;		/*HA 01.10.03 V1.64 new Param for panoadapter*/
	/*V1.95 new array for trolley empty pos*/
		DINT		TrolleyEmptyPositions[MAXTROLLEYS*2]; /*Trick, da 2-dim array nicht geht
														   * wird im Performance nicht gebraucht
														   * hier sind die Leer-Positionen direkt
														   * in den Trolley-Parametern abgelegt,
														   * das ging beim Jet nicht, weil die Kompatibilität
														   ' der Parameter gewahrt bleiben musste (Trolley-Array!)*/
		REAL		MaxTablePosition; /*Enable Position f Feeder runter*/
		REAL		MinTablePosDrop; /*Position des Tisches so, dass Bandrollen mittig unter Saugern sind*/
		REAL		DropOffset;		/* In welchem Abstand soll die Platte an die Stifte gelegt werden? in mm*/
	}Feeder_Param_Typ;

	/* Datenstrukturen für Papierentfernung */
	typedef struct
	{
	/*horizontal*/
		DINT		EnableFeeder;
		DINT		PaperReleaseSingle;
		DINT		PaperReleasePanorama;
		DINT		PaperRemoveLeft;
		DINT		PaperRemoveRight;
		DINT		TrolleyCloseRightStart;		/* Startpos for closing trolley right */
		DINT		TrolleyCloseRightStop;		/* Stoppos for closing trolley right */
		DINT		TrolleyOpenRightStart;		/* Startpos for opening trolley right */
		DINT		TrolleyOpenRightStop;		/* Stoppos for opening trolley right */

		DINT		PaletteDetectStartPos;			/* Startpos for palette detection */
		DINT		PaletteDetectEndPos;  			/* Endpos for palette detection */
		DINT		Reserve1;
		DINT		Reserve2;

	}PaperRemove_Horiz_Pos_Typ;

	typedef struct
	{
	/*vertical*/
		DINT		Up;
		DINT		Down;
		DINT		OnTrolley;
	}PaperRemove_Vert_Pos_Typ;

	typedef struct
	{
	/*speeds*/
		UDINT		TrolleyOpenCloseSpeed;
		UDINT		PaperRemoveSpeed;
	/*times*/
		UDINT		GripOnTime;			/* in 10ms */
		UDINT		GripOffTime;		/* in 10ms */
		PaperRemove_Horiz_Pos_Typ		HorizontalPositions;
		PaperRemove_Vert_Pos_Typ		VerticalPositions;
		UDINT		MaxCurrentDown;
		UDINT		MaxCurrentUp;
		UDINT		PushPos_Horizontal;
		UDINT		PushPos_Vertical;
		UDINT		TrolleyOpenDownSpeed;
		UDINT		TrolleyOpenUpSpeed;
		UDINT		PaperRemoveDownSpeed;
		UDINT		PaperRemoveUpSpeed;
		UDINT		TimeoutOnTrolley;		/* in 10ms */
		UDINT		PaletteDetectSpeed;		/* */
		UDINT		TimeoutUpFromTrolley;	/* in 10ms */
		UDINT		TimeoutOpenTrolleySmall;/* in 10ms */
		UDINT		TimeoutOpenTrolleyBig;	/* in 10ms */
		UDINT		TrolleyDetectSpeed;
		DINT		TrolleyDetectStartPos;
		DINT		TrolleyDetectEndPos;
		USINT		PaperGripCycles;
		DINT		HorPositionPano;		/*HA 01.10.03 V1.64 new Param for panoadapter*/
		DINT		PaperReleasePosVertical;
	}PaperRemove_Param_Typ;

	/*Datenstrukturen für Shuttle*/
	typedef struct
	{
		DINT		EnableFeeder;
		DINT		TakePlate;
		DINT		ReleasePlateMax;
	}Shuttle_Pos_Typ;

	typedef struct
	{
		UDINT		VacuumOnTime;		/* in 10ms */
		UDINT		VacuumOffTime;		/* in 10ms */
		Shuttle_Pos_Typ			Positions;
		REAL DropOffset;
		UDINT		ToAdjusterSpeed;
		UDINT		ToTrolleySpeed;
		REAL		MaxTablePositionDrop;
		BOOL		IgnoreVacuumSwitch;	/*don't check vacuum switch*/
		BOOL		EnablePaperDetection; /*V1.93 Papiersensor schaltbar*/
		DINT		PlateDropPositions[MAXPLATETYPES];
		DINT		ReleasePlatePositions[MAXPLATETYPES]; /*V1.95 Release Posiitons plate-dependant*/
		BOOL		EnablePlateToPaperbasket; /*V2.00 Papiersensor Aktion schaltbar*/
	}Shuttle_Param_Typ;

	/*struct for adjuster Parameter*/
	typedef struct
	{
		UDINT	PinsUpTime;
		UDINT	PinsDownTime;
		UDINT	AdjActiveTime;
		UDINT	AdjInactiveTime;
		UDINT	AdjVacuumOnDelay;
		UDINT	AdjVacuumOffDelay;
		UDINT	TableVacuumOnDelay;
		UDINT	TableVacuumOffDelay;
		UDINT	BlowairOnDelay;
		UDINT	BlowairOffDelay;
		UDINT	TimeoutAdjustedPosition;
		USINT	MaxFailedPlates;
		USINT	MaxAttempts;
		UDINT	AddBlowairValveDelay;
		INT		AdjustSim;
		DINT	FeederAdjustposition; /* vertical position for adjusting */
		DINT	FeederFixposition; /* vertical position for fixing the plate */
	}Adjust_Param_Typ;

	/* struct to hold plate data*/
	typedef struct
	{
		UINT	Number;
		STRING	Name[MAXPLATETYPENAMELENGTH];
		UINT	SeparateBeltTracks;	/*V1.92 separate tracks possible on conveyorbelt*/
		USINT	TurnMode;	/*turn mode for deloader*/
		REAL	XOffset;
		REAL	YOffset;
		REAL	Length;
		REAL	Width;
		REAL	Thickness;
		REAL	Sensitivity;
	/*HA 23.06.03 V1.10*/
	/*Positions for Deloader*/
		UDINT	TakePlatePosition;
		UDINT	ReleasePlatePosition; /* in Performance used for Feeder-horizontal-release-position*/
		UDINT	ReleasePlatePosition2;
		BOOL	Reserve3;
		BOOL	Reserve1;
		INT		Reserve2;
		UDINT	dummy[1];		/*for future enhancements*/
	}Plate_Data_Typ;

	/*struct for global machine data*/
	typedef struct
	{
		STRING	MachineName[32];
		STRING	MachineNumber[6];
		STRING	CustomerName[32];

		REAL	MaxPlateLength;
		REAL	MinPlateLength;
		UDINT	TrolleyRightOffset;
		USINT	TrolleyLeft;
		USINT	TrolleyRight;
		BOOL	AlternatingTrolleys;

		BOOL	XSimulation;
		BOOL	TBSimulation;
		BOOL	ProcessorSimulation;
		BOOL	PunchSimulation;
		BOOL	PaperRemoveEnabled;
		UINT	Language;
		BOOL	Dummy;
		BOOL	FlexibleFeeder;				/*Feeder horizontal present? 1=Yes*/
		BOOL	AutomaticTrolleyOpenClose;
		USINT	reserve1;
		USINT	reserve2;
		USINT	reserve3;
		USINT	reserve4;
		USINT	EnablePaletteLoading;
		USINT	LaserPower;
		UINT 	Resolution;
		UDINT 	ScansPerMinute;
		BOOL	UseOldTiffBlaster;
		USINT	DeloaderTurnStation;		/*deloader turn and positioning station present? 1=hor only, 2=hor+turn*/
	/*neue Var für Laserpower mit Nachkommastelle*/
		UINT	RealLaserPower;
		USINT	MirroredMachine;
		UINT	DisableSlowMode;
		UDINT	SlowModeWaitTime;
	}Global_Data_Typ;

	/*Trolley Data*/
	typedef struct
	{
		STRING 		Name[MAXTROLLEYNAMELENGTH];
		USINT		Number;
		USINT		PlateType;
		BOOL		Empty;				/*Empty flag for single trolley*/
		BOOL		Single;
		BOOL		Double;
		BOOL		NoCover;			/*No cover -> Palette*/
		BOOL		LeftStack;			/*only for double trolley */
		BOOL		RightStack;			/*only for double trolley */
		UINT		PlatesLeft;			/*current Number of plates*/
		UINT		PlatesRight;		/*current Number of plates*/
	/*Positions for OPen / Close*/
		DINT		OpenStart;
		DINT		OpenStop;
		DINT		CloseStart;
		DINT		CloseStop;
	/*Positions for 2-stack trolley*/
		DINT		TakePlateLeft;
		DINT		TakePlateRight;
		DINT		TakePaperLeft;
		DINT		TakePaperRight;
	/* data for Single trolley*/
	/*Positions are stored in "left" data for 2 stack trolley*/

		BOOL		EmptyLeft;		/*double trolley: left stack empty*/
		BOOL		EmptyRight;		/*double trolley: right stack empty*/
		DINT		EmptyPositions[3]; /*Leer Positionen*/
	}Trolley_Data_Typ;

	/*struct for deloader Parameter*/
	typedef struct
	{
		UDINT	PlateTakePosition;
		UDINT	PlateReleasePosition;
		REAL	MinTablePositionTake;
		REAL	MaxTablePositionRelease;
		UDINT	MaxPlateTakePosition;
		UDINT	VacuumOnTime;
		UDINT	VacuumOffTime;
	/*HA 27.01.04 V1.75 Plate length factor for deloading w/out Turnstation*/
		UDINT	PlateLengthAddition; 	/*in mm*/
	/*hor. position to move to for turning (middle)*/
		UDINT	TurnEnabledPosition;
	/*Turn positions in Incr.*/
		UDINT	Turn0Position;
		UDINT	Turn90Position;
		UDINT	Turn180Position;
		DINT	ConveyorBeltSpeed;
		UDINT	TurnSpeed;
		REAL	TableDeloadSpeed;
		REAL	TableDeloadSpeedManual;
		USINT	TurnMode;			/* 0 = no turn, 1 = 90 degrees, 2 = 180 degrees*/
		UDINT	ConveyorBeltDelay;
		REAL	StartTablePosition;	/*Startpos for deloading w/out turnstation*/
		REAL	EndTablePosition;	/*Endpos for deloading w/out turnstation*/
		UDINT	EGMStopDelay;
	/*new for shifted laying off*/
		BOOL	ShiftedLayingOff;
		UDINT	PlateReleasePosition2; /**/
		BOOL	EnableStopPins;
		UDINT	PinsUpDelay;
		UDINT	PinsDownDelay;
		BOOL	SeparateSensors; /*V1.93*/
		UDINT	ConvLateralPulseTime;
		UDINT	ConvLateralMoveTime;
	}Deload_Param_Typ;

	typedef struct
	{
		USINT	TrolleyNumber;
		USINT	PlateType;
		BOOL	TwoStacks;
		USINT	CurrentStack; /*LEFT,RIGHT,DRAWER*/
		USINT	PlateStackInTrolley; /*LEFT,RIGHT,DRAWER*/
		DINT	FeederHorizontalPos;
		DINT	LastStackPos;
		DINT	FeederVerticalPos;
		DINT	PaperRemovePos;
		USINT	LastUsedStack;
	}CurrentDataTyp;

	typedef struct
	{
		UINT	Resolution;
		UINT	LaserPower[MAXPLATETYPES];
	}LaserPowerSettings_Type;

	typedef struct
	{
		BOOL	present; /* a plate is present at that position */
		USINT	PlateType;
		USINT	PlateConfig;
		STRING	FileName[MAXEXPOSEFILENAMELENGTH];
		UINT	ErrorCode;  /* e.g. Paper detected*/
		STRING	ID[JOBIDLENGTH];
		STRING	IDOnDispl[10]; /* weil die ganze ID nicht auf den Schirm passt */
		INT		Status;
		USINT	NextPlateType;
	}PlateInSystem_Type;

	/********************************************************************/
	/* Globale Variablen 												*/
	/********************************************************************/

	/* Struktur als Schnittstelle zur Applikation */
	_GLOBAL	FU_Typ				FU;
	_GLOBAL	X_Param_Typ			X_Param;
	_GLOBAL	Expose_Param_Typ	Expose_Param;

	/*global machine Data*/
	_GLOBAL	Global_Data_Typ	GlobalParameter;

	/*plate data*/
	_GLOBAL	Plate_Data_Typ	PlateTypes[MAXPLATETYPES];
	_GLOBAL	Plate_Data_Typ	PlateParameter;

	_GLOBAL UINT wBildAktuell;
	_GLOBAL UINT wBildNeu;
	_GLOBAL UINT wBildAlt;
	_GLOBAL UINT wBildNr;
	_GLOBAL UINT wBildLast;
	_GLOBAL BOOL xBildExit;
	_GLOBAL BOOL xBildInit;

	_GLOBAL UINT  ACHSE_PIC;
	_GLOBAL UINT  ACHSE_PARAM_PIC;

	_GLOBAL BOOL saveXData;
	_GLOBAL BOOL loadXData;
	_GLOBAL BOOL saveMotorData;
	_GLOBAL BOOL loadMotorData;
	_GLOBAL BOOL saveParameterData;
	_GLOBAL BOOL loadParameterData;

	_GLOBAL BOOL ParkPositionChanged;

	_GLOBAL USINT Cmd[WRITEDATALENGTH];
	_GLOBAL USINT SendMotor;
	_GLOBAL Motor_Typ Motors[MAXMOTORS+1];
	_GLOBAL USINT MotorsConnected;

	_GLOBAL	Trolley_Data_Typ	Trolleys[MAXTROLLEYS];

	/* Strukturen für Funktionseinheiten */
	_GLOBAL	Feeder_Param_Typ		FeederParameter;
	_GLOBAL	PaperRemove_Param_Typ	PaperRemoveParameter;
	_GLOBAL Adjust_Param_Typ		AdjusterParameter;
	_GLOBAL Deload_Param_Typ		DeloaderParameter;
	_GLOBAL	BOOL	OpenTrolleyStart;
	_GLOBAL	BOOL	CloseTrolleyStart;
	_GLOBAL	BOOL	ReferenceStart;
	_GLOBAL	BOOL	PaperRemoveStart;
	_GLOBAL	BOOL	PlateTakingStart;
	_GLOBAL	BOOL	AdjustStart;
	_GLOBAL	BOOL	DeloadStart;
	_GLOBAL	BOOL	ExposeStart;
	_GLOBAL	BOOL	DeloadStart;
	_GLOBAL BOOL	PaperRemoveReady;
	_GLOBAL BOOL	AdjustReady;
	_GLOBAL BOOL	ExposureReady;
	_GLOBAL	BOOL	DeloadReady;

	/* variables for trolley management*/
	_GLOBAL	USINT	CurrentStack;
	_GLOBAL	BOOL	TrolleyRightOpen;
	_GLOBAL	BOOL	TrolleyLeftOpen;
	_GLOBAL	BOOL	TrolleyRightEmpty;
	_GLOBAL	BOOL	TrolleyLeftEmpty;

	/*Sequence controll variabs*/

	_GLOBAL	BOOL	TCPConnected;
	_GLOBAL	USINT	TCPSendCmd;
	_GLOBAL	USINT	TCPCmd[20];
	_GLOBAL	USINT	TCPAnswer[100];
	_GLOBAL	BOOL	TCPRcvFlag;

	_GLOBAL	BOOL	START,AUTO,StartedAutomatically;

	_GLOBAL BOOL	TrolleyEmpty;

	_GLOBAL	BOOL	TrolleyOpen;
	_GLOBAL	BOOL	AlarmBitField[MAXALARMS];
	_GLOBAL	BOOL	AlarmQuitBitField[MAXALARMS];

	_GLOBAL	UINT	AbfrageText1,AbfrageText2,AbfrageText3,AbfrageOK,AbfrageCancel,AbfrageIcon;
	_GLOBAL	UINT	OrgBild,IgnoreButtons,OK_CancelButtonInv,OK_ButtonInv;

	_GLOBAL	USINT	UserLevel;
	_GLOBAL	STRING	FileName[100];
	_GLOBAL	USINT	CounterOn;
	_GLOBAL	UDINT	PlatesToDo;

	_GLOBAL	UINT	PlateType;
	_GLOBAL	BOOL	PanoramaAdapter;

	/*zur Info per TCPIP*/
	_GLOBAL	USINT	SequenceSteps[16];
	_GLOBAL BOOL	PlateTransportSim;
	_GLOBAL STRING  gVERSION[9];
	_GLOBAL DINT AbsMotorPos[MAXMOTORS];
	_GLOBAL REAL AbsMotorPosMm[MAXMOTORS];
	_GLOBAL	CurrentDataTyp	CurrentData;
	_GLOBAL BOOL	StopPlateTaking;
	_GLOBAL BOOL	DisablePaperRemove;
	_GLOBAL	BOOL	StackDetect[2];
	_GLOBAL	BOOL	AlternatingTrolleys;
	_GLOBAL	BOOL	DisableTable;
	_GLOBAL	LaserPowerSettings_Type LaserPowerSettings[MAXLASERPOWERSETTINGS];
	_GLOBAL	BOOL	StatusEGM1;
	_GLOBAL	BOOL	StatusEGM2;
	_GLOBAL	BOOL	SlowMode;
	_GLOBAL USINT	UnexposedPlatesInSystem;
	_GLOBAL BOOL	DataReady;
	_GLOBAL BOOL	ResetStartupSeq;
	_GLOBAL BOOL	DontCloseTrolley;

	_GLOBAL BOOL	BUSY;
	_GLOBAL BOOL	ERROR;
	_GLOBAL BOOL	STANDBY;
	_GLOBAL	BOOL	InEGM1;
	_GLOBAL	BOOL	InEGM2;
	_GLOBAL	BOOL	VCP;
	_GLOBAL UDINT 	PlatesPerHour;
	_GLOBAL	BOOL	BeamON,BeamOFF,TBShutdown;
	_GLOBAL	BOOL 	ParameterChanged;
	_GLOBAL USINT	CANNodeNumber;
	_GLOBAL USINT		gMotorOnDisplay,gSendManSpeeds;

	_GLOBAL PlateInSystem_Type	PlateToDo;
	_GLOBAL PlateInSystem_Type	PlateAtFeeder;
	_GLOBAL PlateInSystem_Type 	PlateAtAdjustedPosition;
	_GLOBAL PlateInSystem_Type	PlateAtDeloader;
	_GLOBAL PlateInSystem_Type	PlateOnConveyorBelt;
	_GLOBAL	Trolley_Data_Typ *pTrolley;
	_GLOBAL	BOOL ManualLoadingStart;
	_GLOBAL	BOOL ManualMode;

#endif
```

### in_out.h
```c
#include <bur\plctypes.h>

/* INPUT */
_GLOBAL	BOOL	In_ServiceMode;
_GLOBAL	BOOL	CoverLockOK;

_GLOBAL	BOOL	In_PaperSensor[2];
_GLOBAL	BOOL	In_FeederHorActive;
_GLOBAL	BOOL	In_FeederHorInactive;
_GLOBAL	BOOL	In_FeederVacuumOK[6];
_GLOBAL	BOOL	In_AdjustVacuumOK[2];

_GLOBAL	BOOL	In_PlateAdjusted[2];
_GLOBAL	BOOL	In_LiftingPinsDown;
_GLOBAL	BOOL	In_ConveyorBeltSensor[2];

_GLOBAL	BOOL	TrolleyCodeSensor;
_GLOBAL	BOOL	BeltLoose;
_GLOBAL	BOOL	DoorsOK;
_GLOBAL	BOOL	In_PaperRemoveUp;

/* evtl für Später, erstmal nicht vorgesehen */
_GLOBAL BOOL	In_VCPOK;
_GLOBAL BOOL	InEGM1;
_GLOBAL BOOL	InEGM2;

/* OUTPUT */
_GLOBAL	BOOL	Out_FeederVacuumOn[6];
_GLOBAL	BOOL	Out_AdjustSuckerActive[3];
_GLOBAL	BOOL	Out_AdjustSuckerVacuumOn[3];
_GLOBAL	BOOL	Out_AdjustSignalCross;
_GLOBAL	BOOL	Out_Horn;    		/*option*/
_GLOBAL	BOOL	Out_PaperGripOn[2];
_GLOBAL BOOL	Out_FeederHorActive;
_GLOBAL	BOOL	Out_ConveyorbeltPinsUp;	/*option*/
_GLOBAL	BOOL	Out_CoverLockOn;		/**/
_GLOBAL	BOOL	Out_ConveyorbeltLateral;
_GLOBAL	BOOL	Out_AdjustPins4and6Up;	/* benötigt für single2*/
_GLOBAL	BOOL	Out_AdjustPin3Up;		/* benötigt für single2 und single quer*/
_GLOBAL	BOOL	Out_AdjustPinsDown;
_GLOBAL	BOOL	Out_LiftingPinsUp;
_GLOBAL	BOOL	Out_LiftingPinsDown;
/* Tischvakuum*/
_GLOBAL	BOOL	AdjustVacuumOn[3];
_GLOBAL	BOOL	AdjustBlowairOn;

/* OUTPUTS */
#ifdef _IN_OUT_C_SRC
_LOCAL BOOL Module4[12];
_LOCAL BOOL Module5[12];
_LOCAL BOOL Module6[12];
#endif
```
